	{attribute 'TcIecLibraryType'}
	{attribute 'external_name' := 'F_VN_SetAt_TcVnRectangle_DINT_GUID_35AC4059_132C_4AEE_E2AA_EA9A3D12C86B'}
	(* Sets the element at the specified index of the container. *)
	FUNCTION F_VN_SetAt_TcVnRectangle_DINT : HRESULT
	VAR_IN_OUT
		stElement	:	TcVnRectangle_DINT;	(* Element to set at the specified container position *)
	END_VAR
	VAR_INPUT
		ipContainer	:	ITcVnContainer;	(* Container with TcVnRectangle_DINT elements, in which the element at position nIndex is replaced by stElement *)
		nIndex	:	ULINT;	(* Index *)
		hrPrev	:	HRESULT;	(* HRESULT indicating the result of previous operations (If SUCCEEDED(hrPrev) equals false, no operation is executed.) *)
	END_VAR

END_FUNCTION

// Functions/Basic Container Operations/F_VN_SetAt/F_VN_SetAt_TcVnVector2_DINT

	{attribute 'TcIecLibraryType'}
	{attribute 'external_name' := 'F_VN_SetAt_TcVnVector2_DINT_GUID_5E02A515_5B29_40CA_DD70_70385858C65C'}
	(* Sets the element at the specified index of the container. *)
	FUNCTION F_VN_SetAt_TcVnVector2_DINT : HRESULT
	VAR_IN_OUT
		aElement	:	TcVnVector2_DINT;	(* Element to set at the specified container position *)
	END_VAR
	VAR_INPUT
		ipContainer	:	ITcVnContainer;	(* Container with TcVnVector2_DINT elements, in which the element at position nIndex is replaced by aElement *)
		nIndex	:	ULINT;	(* Index *)
		hrPrev	:	HRESULT;	(* HRESULT indicating the result of previous operations (If SUCCEEDED(hrPrev) equals false, no operation is executed.) *)
	END_VAR

END_FUNCTION

// Functions/Basic Container Operations/F_VN_SetAt/F_VN_SetAt_TcVnVector2_INT

	{attribute 'TcIecLibraryType'}
	{attribute 'external_name' := 'F_VN_SetAt_TcVnVector2_INT_GUID_9A54C8DF_EFEA_42F1_C006_DE70D5579EDC'}
	(* Sets the element at the specified index of the container. *)
	FUNCTION F_VN_SetAt_TcVnVector2_INT : HRESULT
	VAR_IN_OUT
		aElement	:	TcVnVector2_INT;	(* Element to set at the specified container position *)
	END_VAR
	VAR_INPUT
		ipContainer	:	ITcVnContainer;	(* Container with TcVnVector2_INT elements, in which the element at position nIndex is replaced by aElement *)
		nIndex	:	ULINT;	(* Index *)
		hrPrev	:	HRESULT;	(* HRESULT indicating the result of previous operations (If SUCCEEDED(hrPrev) equals false, no operation is executed.) *)
	END_VAR

END_FUNCTION

// Functions/Basic Container Operations/F_VN_SetAt/F_VN_SetAt_TcVnVector2_REAL

	{attribute 'TcIecLibraryType'}
	{attribute 'external_name' := 'F_VN_SetAt_TcVnVector2_REAL_GUID_8C701179_500E_467C_D95A_AFB507FC193B'}
	(* Sets the element at the specified index of the container. *)
	FUNCTION F_VN_SetAt_TcVnVector2_REAL : HRESULT
	VAR_IN_OUT
		aElement	:	TcVnVector2_REAL;	(* Element to set at the specified container position *)
	END_VAR
	VAR_INPUT
		ipContainer	:	ITcVnContainer;	(* Container with TcVnVector2_REAL elements, in which the element at position nIndex is replaced by aElement *)
		nIndex	:	ULINT;	(* Index *)
		hrPrev	:	HRESULT;	(* HRESULT indicating the result of previous operations (If SUCCEEDED(hrPrev) equals false, no operation is executed.) *)
	END_VAR

END_FUNCTION

// Functions/Basic Container Operations/F_VN_SetAt/F_VN_SetAt_TcVnVector2_SINT

	{attribute 'TcIecLibraryType'}
	{attribute 'external_name' := 'F_VN_SetAt_TcVnVector2_SINT_GUID_41E2A1B6_E23C_4E2B_F5BD_66BD8170D23F'}
	(* Sets the element at the specified index of the container. *)
	FUNCTION F_VN_SetAt_TcVnVector2_SINT : HRESULT
	VAR_IN_OUT
		aElement	:	TcVnVector2_SINT;	(* Element to set at the specified container position *)
	END_VAR
	VAR_INPUT
		ipContainer	:	ITcVnContainer;	(* Container with TcVnVector2_SINT elements, in which the element at position nIndex is replaced by aElement *)
		nIndex	:	ULINT;	(* Index *)
		hrPrev	:	HRESULT;	(* HRESULT indicating the result of previous operations (If SUCCEEDED(hrPrev) equals false, no operation is executed.) *)
	END_VAR

END_FUNCTION

// Functions/Basic Container Operations/F_VN_SetAt/F_VN_SetAt_TcVnVector2_UINT

	{attribute 'TcIecLibraryType'}
	{attribute 'external_name' := 'F_VN_SetAt_TcVnVector2_UINT_GUID_21FE93D3_4D33_43A5_D0AF_B50B4A89EE98'}
	(* Sets the element at the specified index of the container. *)
	FUNCTION F_VN_SetAt_TcVnVector2_UINT : HRESULT
	VAR_IN_OUT
		aElement	:	TcVnVector2_UINT;	(* Element to set at the specified container position *)
	END_VAR
	VAR_INPUT
		ipContainer	:	ITcVnContainer;	(* Container with TcVnVector2_UINT elements, in which the element at position nIndex is replaced by aElement *)
		nIndex	:	ULINT;	(* Index *)
		hrPrev	:	HRESULT;	(* HRESULT indicating the result of previous operations (If SUCCEEDED(hrPrev) equals false, no operation is executed.) *)
	END_VAR

END_FUNCTION

// Functions/Basic Container Operations/F_VN_SetAt/F_VN_SetAt_TcVnVector2_USINT

	{attribute 'TcIecLibraryType'}
	{attribute 'external_name' := 'F_VN_SetAt_TcVnVector2_USINT_GUID_71672D26_1D04_4018_CB62_849B8610E425'}
	(* Sets the element at the specified index of the container. *)
	FUNCTION F_VN_SetAt_TcVnVector2_USINT : HRESULT
	VAR_IN_OUT
		aElement	:	TcVnVector2_USINT;	(* Element to set at the specified container position *)
	END_VAR
	VAR_INPUT
		ipContainer	:	ITcVnContainer;	(* Container with TcVnVector2_USINT elements, in which the element at position nIndex is replaced by aElement *)
		nIndex	:	ULINT;	(* Index *)
		hrPrev	:	HRESULT;	(* HRESULT indicating the result of previous operations (If SUCCEEDED(hrPrev) equals false, no operation is executed.) *)
	END_VAR

END_FUNCTION

// Functions/Basic Container Operations/F_VN_SetAt/F_VN_SetAt_TcVnVector3_INT

	{attribute 'TcIecLibraryType'}
	{attribute 'external_name' := 'F_VN_SetAt_TcVnVector3_INT_GUID_B387FD7B_1A12_472C_FF84_9E1251FBA387'}
	(* Sets the element at the specified index of the container. *)
	FUNCTION F_VN_SetAt_TcVnVector3_INT : HRESULT
	VAR_IN_OUT
		aElement	:	TcVnVector3_INT;	(* Element to set at the specified container position *)
	END_VAR
	VAR_INPUT
		ipContainer	:	ITcVnContainer;	(* Container with TcVnVector3_INT elements, in which the element at position nIndex is replaced by aElement *)
		nIndex	:	ULINT;	(* Index *)
		hrPrev	:	HRESULT;	(* HRESULT indicating the result of previous operations (If SUCCEEDED(hrPrev) equals false, no operation is executed.) *)
	END_VAR

END_FUNCTION

// Functions/Basic Container Operations/F_VN_SetAt/F_VN_SetAt_TcVnVector3_REAL

	{attribute 'TcIecLibraryType'}
	{attribute 'external_name' := 'F_VN_SetAt_TcVnVector3_REAL_GUID_977FE56D_428C_427D_D95B_7AAACF1FD840'}
	(* Sets the element at the specified index of the container. *)
	FUNCTION F_VN_SetAt_TcVnVector3_REAL : HRESULT
	VAR_IN_OUT
		aElement	:	TcVnVector3_REAL;	(* Element to set at the specified container position *)
	END_VAR
	VAR_INPUT
		ipContainer	:	ITcVnContainer;	(* Container with TcVnVector3_REAL elements, in which the element at position nIndex is replaced by aElement *)
		nIndex	:	ULINT;	(* Index *)
		hrPrev	:	HRESULT;	(* HRESULT indicating the result of previous operations (If SUCCEEDED(hrPrev) equals false, no operation is executed.) *)
	END_VAR

END_FUNCTION

// Functions/Basic Container Operations/F_VN_SetAt/F_VN_SetAt_TcVnVector3_SINT

	{attribute 'TcIecLibraryType'}
	{attribute 'external_name' := 'F_VN_SetAt_TcVnVector3_SINT_GUID_82C45DC0_A60E_4C50_ED24_B824FCF78FFB'}
	(* Sets the element at the specified index of the container. *)
	FUNCTION F_VN_SetAt_TcVnVector3_SINT : HRESULT
	VAR_IN_OUT
		aElement	:	TcVnVector3_SINT;	(* Element to set at the specified container position *)
	END_VAR
	VAR_INPUT
		ipContainer	:	ITcVnContainer;	(* Container with TcVnVector3_SINT elements, in which the element at position nIndex is replaced by aElement *)
		nIndex	:	ULINT;	(* Index *)
		hrPrev	:	HRESULT;	(* HRESULT indicating the result of previous operations (If SUCCEEDED(hrPrev) equals false, no operation is executed.) *)
	END_VAR

END_FUNCTION

// Functions/Basic Container Operations/F_VN_SetAt/F_VN_SetAt_TcVnVector3_UINT

	{attribute 'TcIecLibraryType'}
	{attribute 'external_name' := 'F_VN_SetAt_TcVnVector3_UINT_GUID_B07401BC_3104_41A1_CD0F_B943A0C58B6B'}
	(* Sets the element at the specified index of the container. *)
	FUNCTION F_VN_SetAt_TcVnVector3_UINT : HRESULT
	VAR_IN_OUT
		aElement	:	TcVnVector3_UINT;	(* Element to set at the specified container position *)
	END_VAR
	VAR_INPUT
		ipContainer	:	ITcVnContainer;	(* Container with TcVnVector3_UINT elements, in which the element at position nIndex is replaced by aElement *)
		nIndex	:	ULINT;	(* Index *)
		hrPrev	:	HRESULT;	(* HRESULT indicating the result of previous operations (If SUCCEEDED(hrPrev) equals false, no operation is executed.) *)
	END_VAR

END_FUNCTION

// Functions/Basic Container Operations/F_VN_SetAt/F_VN_SetAt_TcVnVector3_USINT

	{attribute 'TcIecLibraryType'}
	{attribute 'external_name' := 'F_VN_SetAt_TcVnVector3_USINT_GUID_CA981836_58FF_4571_CBB8_6E1A27874793'}
	(* Sets the element at the specified index of the container. *)
	FUNCTION F_VN_SetAt_TcVnVector3_USINT : HRESULT
	VAR_IN_OUT
		aElement	:	TcVnVector3_USINT;	(* Element to set at the specified container position *)
	END_VAR
	VAR_INPUT
		ipContainer	:	ITcVnContainer;	(* Container with TcVnVector3_USINT elements, in which the element at position nIndex is replaced by aElement *)
		nIndex	:	ULINT;	(* Index *)
		hrPrev	:	HRESULT;	(* HRESULT indicating the result of previous operations (If SUCCEEDED(hrPrev) equals false, no operation is executed.) *)
	END_VAR

END_FUNCTION

// Functions/Basic Container Operations/F_VN_SetAt/F_VN_SetAt_TcVnVector4_DINT

	{attribute 'TcIecLibraryType'}
	{attribute 'external_name' := 'F_VN_SetAt_TcVnVector4_DINT_GUID_84075105_DF73_46B7_C61E_1F0647F1D871'}
	(* Sets the element at the specified index of the container. *)
	FUNCTION F_VN_SetAt_TcVnVector4_DINT : HRESULT
	VAR_IN_OUT
		aElement	:	TcVnVector4_DINT;	(* Element to set at the specified container position *)
	END_VAR
	VAR_INPUT
		ipContainer	:	ITcVnContainer;	(* Container with TcVnVector4_DINT elements, in which the element at position nIndex is replaced by aElement *)
		nIndex	:	ULINT;	(* Index *)
		hrPrev	:	HRESULT;	(* HRESULT indicating the result of previous operations (If SUCCEEDED(hrPrev) equals false, no operation is executed.) *)
	END_VAR

END_FUNCTION

// Functions/Basic Container Operations/F_VN_SetAt/F_VN_SetAt_TcVnVector4_INT

	{attribute 'TcIecLibraryType'}
	{attribute 'external_name' := 'F_VN_SetAt_TcVnVector4_INT_GUID_4C86CA39_B19A_4E94_C5DE_D1DC020F94C8'}
	(* Sets the element at the specified index of the container. *)
	FUNCTION F_VN_SetAt_TcVnVector4_INT : HRESULT
	VAR_IN_OUT
		aElement	:	TcVnVector4_INT;	(* Element to set at the specified container position *)
	END_VAR
	VAR_INPUT
		ipContainer	:	ITcVnContainer;	(* Container with TcVnVector4_INT elements, in which the element at position nIndex is replaced by aElement *)
		nIndex	:	ULINT;	(* Index *)
		hrPrev	:	HRESULT;	(* HRESULT indicating the result of previous operations (If SUCCEEDED(hrPrev) equals false, no operation is executed.) *)
	END_VAR

END_FUNCTION

// Functions/Basic Container Operations/F_VN_SetAt/F_VN_SetAt_TcVnVector4_LREAL

	{attribute 'TcIecLibraryType'}
	{attribute 'external_name' := 'F_VN_SetAt_TcVnVector4_LREAL_GUID_B3814A00_38B2_4F72_CE05_8FB87EDAF63D'}
	(* Sets the element at the specified index of the container. *)
	FUNCTION F_VN_SetAt_TcVnVector4_LREAL : HRESULT
	VAR_IN_OUT
		aElement	:	TcVnVector4_LREAL;	(* Element to set at the specified container position *)
	END_VAR
	VAR_INPUT
		ipContainer	:	ITcVnContainer;	(* Container with TcVnVector4_LREAL elements, in which the element at position nIndex is replaced by aElement *)
		nIndex	:	ULINT;	(* Index *)
		hrPrev	:	HRESULT;	(* HRESULT indicating the result of previous operations (If SUCCEEDED(hrPrev) equals false, no operation is executed.) *)
	END_VAR

END_FUNCTION

// Functions/Basic Container Operations/F_VN_SetAt/F_VN_SetAt_TcVnVector4_REAL

	{attribute 'TcIecLibraryType'}
	{attribute 'external_name' := 'F_VN_SetAt_TcVnVector4_REAL_GUID_64AEDC0F_5778_44DB_ECE6_E811B6DE732F'}
	(* Sets the element at the specified index of the container. *)
	FUNCTION F_VN_SetAt_TcVnVector4_REAL : HRESULT
	VAR_IN_OUT
		aElement	:	TcVnVector4_REAL;	(* Element to set at the specified container position *)
	END_VAR
	VAR_INPUT
		ipContainer	:	ITcVnContainer;	(* Container with TcVnVector4_REAL elements, in which the element at position nIndex is replaced by aElement *)
		nIndex	:	ULINT;	(* Index *)
		hrPrev	:	HRESULT;	(* HRESULT indicating the result of previous operations (If SUCCEEDED(hrPrev) equals false, no operation is executed.) *)
	END_VAR

END_FUNCTION

// Functions/Basic Container Operations/F_VN_SetAt/F_VN_SetAt_TcVnVector4_SINT

	{attribute 'TcIecLibraryType'}
	{attribute 'external_name' := 'F_VN_SetAt_TcVnVector4_SINT_GUID_9A249CC5_D1EE_48B3_F4D3_D6345D13532B'}
	(* Sets the element at the specified index of the container. *)
	FUNCTION F_VN_SetAt_TcVnVector4_SINT : HRESULT
	VAR_IN_OUT
		aElement	:	TcVnVector4_SINT;	(* Element to set at the specified container position *)
	END_VAR
	VAR_INPUT
		ipContainer	:	ITcVnContainer;	(* Container with TcVnVector4_SINT elements, in which the element at position nIndex is replaced by aElement *)
		nIndex	:	ULINT;	(* Index *)
		hrPrev	:	HRESULT;	(* HRESULT indicating the result of previous operations (If SUCCEEDED(hrPrev) equals false, no operation is executed.) *)
	END_VAR

END_FUNCTION

// Functions/Basic Container Operations/F_VN_SetAt/F_VN_SetAt_TcVnVector4_UINT

	{attribute 'TcIecLibraryType'}
	{attribute 'external_name' := 'F_VN_SetAt_TcVnVector4_UINT_GUID_9C7C3011_85A8_431A_EEDE_04346BDEC621'}
	(* Sets the element at the specified index of the container. *)
	FUNCTION F_VN_SetAt_TcVnVector4_UINT : HRESULT
	VAR_IN_OUT
		aElement	:	TcVnVector4_UINT;	(* Element to set at the specified container position *)
	END_VAR
	VAR_INPUT
		ipContainer	:	ITcVnContainer;	(* Container with TcVnVector4_UINT elements, in which the element at position nIndex is replaced by aElement *)
		nIndex	:	ULINT;	(* Index *)
		hrPrev	:	HRESULT;	(* HRESULT indicating the result of previous operations (If SUCCEEDED(hrPrev) equals false, no operation is executed.) *)
	END_VAR

END_FUNCTION

// Functions/Basic Container Operations/F_VN_SetAt/F_VN_SetAt_TcVnVector4_USINT

	{attribute 'TcIecLibraryType'}
	{attribute 'external_name' := 'F_VN_SetAt_TcVnVector4_USINT_GUID_8CCBCF1A_6BF1_414F_D7CE_FA6418BF3A5A'}
	(* Sets the element at the specified index of the container. *)
	FUNCTION F_VN_SetAt_TcVnVector4_USINT : HRESULT
	VAR_IN_OUT
		aElement	:	TcVnVector4_USINT;	(* Element to set at the specified container position *)
	END_VAR
	VAR_INPUT
		ipContainer	:	ITcVnContainer;	(* Container with TcVnVector4_USINT elements, in which the element at position nIndex is replaced by aElement *)
		nIndex	:	ULINT;	(* Index *)
		hrPrev	:	HRESULT;	(* HRESULT indicating the result of previous operations (If SUCCEEDED(hrPrev) equals false, no operation is executed.) *)
	END_VAR

END_FUNCTION

// Functions/Basic Container Operations/F_VN_SetAt/F_VN_SetAt_UDINT

	{attribute 'TcIecLibraryType'}
	{attribute 'external_name' := 'F_VN_SetAt_UDINT_GUID_C39B4E59_D3B2_44DA_C04B_593E8FE83763'}
	(* Sets the element at the specified index of the container. *)
	FUNCTION F_VN_SetAt_UDINT : HRESULT
	VAR_INPUT
		nElement	:	UDINT;	(* Element to set at the specified container position *)
		ipContainer	:	ITcVnContainer;	(* Container with UDINT elements, in which the element at position nIndex is replaced by nElement *)
		nIndex	:	ULINT;	(* Index *)
		hrPrev	:	HRESULT;	(* HRESULT indicating the result of previous operations (If SUCCEEDED(hrPrev) equals false, no operation is executed.) *)
	END_VAR

END_FUNCTION

// Functions/Basic Container Operations/F_VN_SetAt/F_VN_SetAt_UINT

	{attribute 'TcIecLibraryType'}
	{attribute 'external_name' := 'F_VN_SetAt_UINT_GUID_973D05B9_94F7_4B2D_E393_23B939525C18'}
	(* Sets the element at the specified index of the container. *)
	FUNCTION F_VN_SetAt_UINT : HRESULT
	VAR_INPUT
		nElement	:	UINT;	(* Element to set at the specified container position *)
		ipContainer	:	ITcVnContainer;	(* Container with UINT elements, in which the element at position nIndex is replaced by nElement *)
		nIndex	:	ULINT;	(* Index *)
		hrPrev	:	HRESULT;	(* HRESULT indicating the result of previous operations (If SUCCEEDED(hrPrev) equals false, no operation is executed.) *)
	END_VAR

END_FUNCTION

// Functions/Basic Container Operations/F_VN_SetAt/F_VN_SetAt_ULINT

	{attribute 'TcIecLibraryType'}
	{attribute 'external_name' := 'F_VN_SetAt_ULINT_GUID_FC881A2A_C368_47AC_FDE8_4603A11A5BED'}
	(* Sets the element at the specified index of the container. *)
	FUNCTION F_VN_SetAt_ULINT : HRESULT
	VAR_INPUT
		nElement	:	ULINT;	(* Element to set at the specified container position *)
		ipContainer	:	ITcVnContainer;	(* Container with ULINT elements, in which the element at position nIndex is replaced by nElement *)
		nIndex	:	ULINT;	(* Index *)
		hrPrev	:	HRESULT;	(* HRESULT indicating the result of previous operations (If SUCCEEDED(hrPrev) equals false, no operation is executed.) *)
	END_VAR

END_FUNCTION

// Functions/Basic Container Operations/F_VN_SetAt/F_VN_SetAt_USINT

	{attribute 'TcIecLibraryType'}
	{attribute 'external_name' := 'F_VN_SetAt_USINT_GUID_71675C04_000B_40FA_E123_CBE4050ACA90'}
	(* Sets the element at the specified index of the container. *)
	FUNCTION F_VN_SetAt_USINT : HRESULT
	VAR_INPUT
		nElement	:	USINT;	(* Element to set at the specified container position *)
		ipContainer	:	ITcVnContainer;	(* Container with USINT elements, in which the element at position nIndex is replaced by nElement *)
		nIndex	:	ULINT;	(* Index *)
		hrPrev	:	HRESULT;	(* HRESULT indicating the result of previous operations (If SUCCEEDED(hrPrev) equals false, no operation is executed.) *)
	END_VAR

END_FUNCTION

// Functions/Geometric and Coordinate Transformations/Calibration/F_VN_CalibrateCamera

	{attribute 'TcIecLibraryType'}
	{attribute 'external_name' := 'F_VN_CalibrateCamera_GUID_EBB15309_7B02_4BBD_EDF8_3E60282ECCFA'}
	(* Compute the camera parameters (intrinsic + extrinsic) by evaluating an image containing a calibration pattern (circles). *)
	FUNCTION F_VN_CalibrateCamera : HRESULT
	VAR_INPUT
		ipSrcImage	:	ITcVnImage;	(* Source image containing a calibration pattern (1 channel, USINT elements) *)
		ipReferencePoints	:	ITcVnContainer;	(* Reference calibration pattern point positions (ContainerType_Vector_TcVnPoint3_REAL) *)
	END_VAR
	VAR_IN_OUT
		aCameraMatrix	:	TcVnMatrix3x3_LREAL;	(* Returns the camera matrix *)
		aDistortionCoefficients	:	TcVnArray8_LREAL;	(* Returns the lens distortion coefficients [k1, k2, p1, p2, k3, k4, k5, k6] *)
		aRotationMatrix	:	TcVnMatrix3x3_LREAL;	(* Returns the rotation matrix *)
		aTranslationVector	:	TcVnVector3_LREAL;	(* Returns the translation vector *)
		fReprojError	:	LREAL;	(* Returns the reprojection error *)
		stBlobDetectionParams	:	TcVnParamsBlobDetection;	(* Parameters for the internally used F_VN_DetectBlobs function *)
		stCalibrationOptions	:	TcVnCameraCalibrationOptions;	(* Calibration options *)
	END_VAR
	VAR_INPUT
		hrPrev	:	HRESULT;	(* HRESULT indicating the result of previous operations (If SUCCEEDED(hrPrev) equals false, no operation is executed.) *)
	END_VAR

END_FUNCTION

// Functions/Geometric and Coordinate Transformations/Calibration/F_VN_CalibrateCameraExp

	{attribute 'TcIecLibraryType'}
	{attribute 'external_name' := 'F_VN_CalibrateCameraExp_GUID_1D6493E0_8C99_44E7_F620_1AFFF7BB97DC'}
	(* Compute the camera parameters (intrinsic + extrinsic) by evaluating images containing a calibration pattern (circles). The extrinsic parameters are computed for the first image in the array. (expert function) *)
	FUNCTION F_VN_CalibrateCameraExp : HRESULT
	VAR_INPUT
		pSrcImages	:	PVOID;	(* Pointer to an array of source images, each containing the same calibration pattern (1 channel, USINT elements) *)
		nSrcArraySize	:	UINT;	(* pSrcImages array size *)
		ipReferencePoints	:	ITcVnContainer;	(* Reference calibration pattern point positions (ContainerType_Vector_TcVnPoint3_REAL) *)
	END_VAR
	VAR_IN_OUT
		aCameraMatrix	:	TcVnMatrix3x3_LREAL;	(* Returns the camera matrix *)
		aDistortionCoefficients	:	TcVnArray8_LREAL;	(* Returns the lens distortion coefficients [k1, k2, p1, p2, k3, k4, k5, k6] *)
		aRotationMatrix	:	TcVnMatrix3x3_LREAL;	(* Returns the rotation matrix *)
		aTranslationVector	:	TcVnVector3_LREAL;	(* Returns the translation vector *)
		fReprojError	:	LREAL;	(* Returns the reprojection error *)
		stBlobDetectionParams	:	TcVnParamsBlobDetection;	(* Parameters for the internally used F_VN_DetectBlobs function *)
		stCalibrationOptions	:	TcVnCameraCalibrationOptions;	(* Calibration options *)
	END_VAR
	VAR_INPUT
		hrPrev	:	HRESULT;	(* HRESULT indicating the result of previous operations (If SUCCEEDED(hrPrev) equals false, no operation is executed.) *)
	END_VAR

END_FUNCTION

// Functions/Geometric and Coordinate Transformations/Calibration/F_VN_CalibrateCameraExp2

	{attribute 'TcIecLibraryType'}
	{attribute 'external_name' := 'F_VN_CalibrateCameraExp2_GUID_8981380C_F1D9_4601_D366_FF624EB09033'}
	(* Compute the camera parameters (intrinsic + extrinsic) by evaluating images containing a calibration pattern (circles). The extrinsic parameters are computed for the first image in the array. (expert function) *)
	FUNCTION F_VN_CalibrateCameraExp2 : HRESULT
	VAR_INPUT
		pSrcImages	:	PVOID;	(* Pointer to an array of source images, each containing the same calibration pattern (1 channel, USINT elements) *)
		nSrcArraySize	:	UINT;	(* pSrcImages array size *)
		ipReferencePoints	:	ITcVnContainer;	(* Reference calibration pattern point positions (ContainerType_Vector_TcVnPoint3_REAL) *)
	END_VAR
	VAR_IN_OUT
		aCameraMatrix	:	TcVnMatrix3x3_LREAL;	(* Returns the camera matrix *)
		aDistortionCoefficients	:	TcVnArray8_LREAL;	(* Returns the lens distortion coefficients [k1, k2, p1, p2, k3, k4, k5, k6] *)
		aRotationMatrix	:	TcVnMatrix3x3_LREAL;	(* Returns the rotation matrix *)
		aTranslationVector	:	TcVnVector3_LREAL;	(* Returns the translation vector *)
		fReprojError	:	LREAL;	(* Returns the reprojection error *)
		stBlobDetectionParams	:	TcVnParamsBlobDetection;	(* Parameters for the internally used F_VN_DetectBlobs function *)
		stCalibrationOptions	:	TcVnCameraCalibrationOptions;	(* Calibration options *)
	END_VAR
	VAR_INPUT
		bSubpixelAccuracy	:	BOOL;	(* If true, the pattern points are detected with subpixel accuracy *)
		eEdgeDirection	:	ETcVnEdgeDirection;	(* Specification of the edge direction to search for (from center to outside ellipse) *)
		fMinStrength	:	REAL;	(* Specification of the minimum strength (intensity difference) of the edge to search for *)
		nMaxThickness	:	UDINT;	(* Specification of the maximum thickness of the edge to search for, which means fMinStrength must be reached within nMaxThickness pixels *)
		nSubpixelsIterations	:	UDINT;	(* Specifies the number of subpixels (for INTERPOLATION, 10 - 20 usually is sufficient) or maximum number of iterations for optimizing the parameters (for APPROX_ERF and APPROX_GAUSSIAN, 50 - 100 usually is sufficient) *)
		nSearchLines	:	UDINT;	(* Specifies the amount of search lines, which are equally distributed in all directions (must be >= 8 and a multiple of 4) *)
		fApproxPrecision	:	REAL;	(* Specifies the approximation precision for APPROX_ERF and APPROX_GAUSSIAN (0.001 usually is sufficient, unused for INTERPOLATION) *)
		eAlgorithm	:	ETcVnEdgeDetectionAlgorithm;	(* Selection of the edge detection algorithm *)
		hrPrev	:	HRESULT;	(* HRESULT indicating the result of previous operations (If SUCCEEDED(hrPrev) equals false, no operation is executed.) *)
	END_VAR

END_FUNCTION

// Functions/Geometric and Coordinate Transformations/Calibration/F_VN_CalibrateCameraExp3

	{attribute 'TcIecLibraryType'}
	{attribute 'external_name' := 'F_VN_CalibrateCameraExp3_GUID_D9F3CD5D_1398_4870_FF18_533CD0366399'}
	(* Compute the camera parameters (intrinsic + extrinsic) by evaluating images containing a calibration pattern (circles). The extrinsic parameters are computed for the first image in the array. (expert function) *)
	FUNCTION F_VN_CalibrateCameraExp3 : HRESULT
	VAR_INPUT
		pSrcImages	:	PVOID;	(* Pointer to an array of source images, each containing the same calibration pattern (1 channel, USINT elements) *)
		nSrcArraySize	:	UINT;	(* pSrcImages array size *)
		ipReferencePoints	:	ITcVnContainer;	(* Reference calibration pattern point positions (ContainerType_Vector_TcVnPoint3_REAL) *)
	END_VAR
	VAR_IN_OUT
		aCameraMatrix	:	TcVnMatrix3x3_LREAL;	(* Returns the camera matrix *)
		aDistortionCoefficients	:	TcVnArray8_LREAL;	(* Returns the lens distortion coefficients [k1, k2, p1, p2, k3, k4, k5, k6] *)
		aRotationMatrix	:	TcVnMatrix3x3_LREAL;	(* Returns the rotation matrix *)
		aTranslationVector	:	TcVnVector3_LREAL;	(* Returns the translation vector *)
		fReprojError	:	LREAL;	(* Returns the reprojection error *)
		stBlobDetectionParams	:	TcVnParamsBlobDetection;	(* Parameters for the internally used F_VN_DetectBlobs function *)
		stCalibrationOptions	:	TcVnCameraCalibrationOptions;	(* Calibration options *)
	END_VAR
	VAR_INPUT
		bSubpixelAccuracy	:	BOOL;	(* If true, the pattern points are detected with subpixel accuracy *)
		eEdgeDirection	:	ETcVnEdgeDirection;	(* Specification of the edge direction to search for (from center to outside ellipse) *)
		fMinStrength	:	REAL;	(* Specification of the minimum strength (intensity difference) of the edge to search for *)
		nMaxThickness	:	UDINT;	(* Specification of the maximum thickness of the edge to search for, which means fMinStrength must be reached within nMaxThickness pixels *)
		nSubpixelsIterations	:	UDINT;	(* Specifies the number of subpixels (for INTERPOLATION, 10 - 20 usually is sufficient) or maximum number of iterations for optimizing the parameters (for APPROX_ERF and APPROX_GAUSSIAN, 50 - 100 usually is sufficient) *)
		nSearchLines	:	UDINT;	(* Specifies the amount of search lines, which are equally distributed in all directions (must be >= 8 and a multiple of 4) *)
		fApproxPrecision	:	REAL;	(* Specifies the approximation precision for APPROX_ERF and APPROX_GAUSSIAN (0.001 usually is sufficient, unused for INTERPOLATION) *)
		eAlgorithm	:	ETcVnEdgeDetectionAlgorithm;	(* Selection of the edge detection algorithm *)
		eWorldSystem	:	ETcVnWorldCoordinateSystem;	(* World coordinate system orientation *)
		hrPrev	:	HRESULT;	(* HRESULT indicating the result of previous operations (If SUCCEEDED(hrPrev) equals false, no operation is executed.) *)
	END_VAR

END_FUNCTION

// Functions/Geometric and Coordinate Transformations/Calibration/F_VN_CalibrateCameraManually

	{attribute 'TcIecLibraryType'}
	{attribute 'external_name' := 'F_VN_CalibrateCameraManually_GUID_5DA30166_3B16_4F1A_EA40_4DD63022F860'}
	(* Compute the camera parameters (intrinsic + extrinsic). The extrinsic parameters are computed for the first inner container. *)
	FUNCTION F_VN_CalibrateCameraManually : HRESULT
	VAR_INPUT
		ipImagePoints	:	ITcVnContainer;	(* Provided image points of multiple images (ContainerType_Vector_Vector_TcVnPoint2_REAL, each inner container with at least 6 points). The container and point order must match ipReferencePoints. *)
		nImageWidth	:	UDINT;	(* Image width *)
		nImageHeight	:	UDINT;	(* Image height *)
		ipReferencePoints	:	ITcVnContainer;	(* Reference world points (ContainerType_Vector_Vector_TcVnPoint3_REAL). The number of inner containers and their amount of points must match ipImagePoints. *)
	END_VAR
	VAR_IN_OUT
		aCameraMatrix	:	TcVnMatrix3x3_LREAL;	(* Returns the camera matrix *)
		aDistortionCoefficients	:	TcVnArray8_LREAL;	(* Returns the lens distortion coefficients [k1, k2, p1, p2, k3, k4, k5, k6] *)
		aRotationMatrix	:	TcVnMatrix3x3_LREAL;	(* Returns the rotation matrix (for the first inner container) *)
		aTranslationVector	:	TcVnVector3_LREAL;	(* Returns the translation vector (for the first inner container) *)
		fReprojError	:	LREAL;	(* Returns the reprojection error *)
		stCalibrationOptions	:	TcVnCameraCalibrationOptions;	(* Calibration options *)
	END_VAR
	VAR_INPUT
		hrPrev	:	HRESULT;	(* HRESULT indicating the result of previous operations (If SUCCEEDED(hrPrev) equals false, no operation is executed.) *)
	END_VAR

END_FUNCTION

// Functions/Geometric and Coordinate Transformations/Calibration/F_VN_CalibrateCameraManuallyExp

	{attribute 'TcIecLibraryType'}
	{attribute 'external_name' := 'F_VN_CalibrateCameraManuallyExp_GUID_DECD6B85_89B7_4630_E66B_3B96B0529CB2'}
	(* Compute the camera parameters (intrinsic + extrinsic). The extrinsic parameters are computed for the first inner container. (expert function) *)
	FUNCTION F_VN_CalibrateCameraManuallyExp : HRESULT
	VAR_INPUT
		ipImagePoints	:	ITcVnContainer;	(* Provided image points of multiple images (ContainerType_Vector_Vector_TcVnPoint2_REAL, each inner container with at least 6 points). The container and point order must match ipReferencePoints. *)
		nImageWidth	:	UDINT;	(* Image width *)
		nImageHeight	:	UDINT;	(* Image height *)
		ipReferencePoints	:	ITcVnContainer;	(* Reference world points (ContainerType_Vector_Vector_TcVnPoint3_REAL). The number of inner containers and their amount of points must match ipImagePoints. *)
	END_VAR
	VAR_IN_OUT
		aCameraMatrix	:	TcVnMatrix3x3_LREAL;	(* Returns the camera matrix *)
		aDistortionCoefficients	:	TcVnArray8_LREAL;	(* Returns the lens distortion coefficients [k1, k2, p1, p2, k3, k4, k5, k6] *)
		aRotationMatrix	:	TcVnMatrix3x3_LREAL;	(* Returns the rotation matrix (for the first inner container) *)
		aTranslationVector	:	TcVnVector3_LREAL;	(* Returns the translation vector (for the first inner container) *)
		fReprojError	:	LREAL;	(* Returns the reprojection error *)
		stCalibrationOptions	:	TcVnCameraCalibrationOptions;	(* Calibration options *)
	END_VAR
	VAR_INPUT
		eWorldSystem	:	ETcVnWorldCoordinateSystem;	(* World coordinate system orientation *)
		hrPrev	:	HRESULT;	(* HRESULT indicating the result of previous operations (If SUCCEEDED(hrPrev) equals false, no operation is executed.) *)
	END_VAR

END_FUNCTION

// Functions/Geometric and Coordinate Transformations/Calibration/F_VN_CalibrateCameraPlanar

	{attribute 'TcIecLibraryType'}
	{attribute 'external_name' := 'F_VN_CalibrateCameraPlanar_GUID_DD8D0D8C_ACE8_4133_C290_06DF72655118'}
	(* Calibrate camera using a planar calibration pattern comprised of four circles marking the corners of a rectangle. *)
	FUNCTION F_VN_CalibrateCameraPlanar : HRESULT
	VAR_INPUT
		ipSrcImage	:	ITcVnImage;	(* Binary source image (background zero, markers non-zero) *)
	END_VAR
	VAR_IN_OUT
		aMarkerPositions	:	TcVnArray4_Point2_REAL;	(* Marker positions within their plane using world units (right-handed coordinate system) *)
		aTransformationMatrix	:	TcVnMatrix3x3_LREAL;	(* Returns a 3-by-3 matrix for the transformation from image coordinates into the reference coordinate system *)
	END_VAR
	VAR_INPUT
		hrPrev	:	HRESULT;	(* HRESULT indicating the result of previous operations (If SUCCEEDED(hrPrev) equals false, no operation is executed.) *)
	END_VAR

END_FUNCTION

// Functions/Geometric and Coordinate Transformations/Calibration/F_VN_CalibrateCameraPlanarExp

	{attribute 'TcIecLibraryType'}
	{attribute 'external_name' := 'F_VN_CalibrateCameraPlanarExp_GUID_7DEAD94E_63B2_4C34_D746_EB385A5F99A0'}
	(* Calibrate camera using a planar calibration pattern comprised of four circles marking the corners of a rectangle. (expert function) *)
	FUNCTION F_VN_CalibrateCameraPlanarExp : HRESULT
	VAR_INPUT
		ipSrcImage	:	ITcVnImage;	(* Binary source image (background zero, markers non-zero) *)
	END_VAR
	VAR_IN_OUT
		aMarkerPositions	:	TcVnArray4_Point2_REAL;	(* Marker positions within their plane using world units (right-handed coordinate system) *)
		aTransformationMatrix	:	TcVnMatrix3x3_LREAL;	(* Returns a 3-by-3 matrix for the transformation from image coordinates into the reference coordinate system *)
		aMarkerImagePositions	:	TcVnArray4_Point2_REAL;	(* Returns the marker positions in image coordinates (left-handed coordinate system) *)
	END_VAR
	VAR_INPUT
		nMinMarkerArea	:	UDINT;	(* Minimum area for the detection of markers (Smaller markers are ignored.) *)
		nMaxMarkerArea	:	UDINT;	(* Maximum area for the detection of markers (Larger markers are ignored.) *)
		fMaxMarkerEccentricity	:	LREAL;	(* Maximum eccenticity for the detection of markers (The eccentricity measures deviations from a round shape (eccentricity = 0: round object; eccentricity = 1.0:  linear object).) *)
		hrPrev	:	HRESULT;	(* HRESULT indicating the result of previous operations (If SUCCEEDED(hrPrev) equals false, no operation is executed.) *)
	END_VAR

END_FUNCTION

// Functions/Geometric and Coordinate Transformations/Calibration/F_VN_CalibrateLinescanCamera

	{attribute 'TcIecLibraryType'}
	{attribute 'external_name' := 'F_VN_CalibrateLinescanCamera_GUID_800BBE18_64E6_4C93_C932_85B991825405'}
	(* Compute the camera parameters (intrinsic + extrinsic) by evaluating images containing a line calibration pattern. The pattern must consist of alternating vertical and diagonal lines, with each diagonal having the same constant slope: |\|\|...\|. The results are only valid for the x-direction of a line scan image. To get accurate x-values for a transformation into world coordinates, the y-coordinate must be set to half the sensor width and so equal to the cy-value of the camera matrix. For other y-values, the results are approximated and can be inaccurate. The extrinsic parameters are computed for the first image in the array. *)
	FUNCTION F_VN_CalibrateLinescanCamera : HRESULT
	VAR_INPUT
		pSrcImages	:	PVOID;	(* Pointer to an array of 1 or more source images (1 channel). If the images have more than 1 row, each row must contain an image of the same pattern position. *)
		nSrcArraySize	:	UINT;	(* pSrcImages array size *)
		ipPatternLineOrigins	:	ITcVnContainer;	(* X position of the pattern line origins (ContainerType_Vector_REAL, usually same origin for vertical and following diagonal line) *)
		fSlopeRad	:	LREAL;	(* Slope of the diagonal line in rad (> 0, < PI/2), relative to the vertical line (i.e., 0 would be a vertical line, PI/2 a horizontal line) *)
	END_VAR
	VAR_IN_OUT
		aCameraMatrix	:	TcVnMatrix3x3_LREAL;	(* Returns the camera matrix *)
		aDistortionCoefficients	:	TcVnArray8_LREAL;	(* Returns the lens distortion coefficients [k1, k2, p1, p2, k3, k4, k5, k6] *)
		aRotationMatrix	:	TcVnMatrix3x3_LREAL;	(* Returns the rotation matrix *)
		aTranslationVector	:	TcVnVector3_LREAL;	(* Returns the translation vector *)
		fReprojError	:	LREAL;	(* Returns the reprojection error *)
		stCalibrationOptions	:	TcVnCameraCalibrationOptions;	(* Calibration options (recommended to set bFixAspectRatio, bFixPrincipalPoint, bZeroTangentDist) *)
	END_VAR
	VAR_INPUT
		eEdgeDirection	:	ETcVnEdgeDirection;	(* Specification of the edge direction to search for *)
		hrPrev	:	HRESULT;	(* HRESULT indicating the result of previous operations (If SUCCEEDED(hrPrev) equals false, no operation is executed.) *)
	END_VAR

END_FUNCTION

// Functions/Geometric and Coordinate Transformations/Calibration/F_VN_CalibrateLinescanCameraExp

	{attribute 'TcIecLibraryType'}
	{attribute 'external_name' := 'F_VN_CalibrateLinescanCameraExp_GUID_AD67159F_52AC_4940_E181_6CB9805B9B64'}
	(* Compute the camera parameters (intrinsic + extrinsic) by evaluating images containing a line calibration pattern. The pattern must consist of alternating vertical and diagonal lines, with each diagonal having the same constant slope: |\|\|...\|. The results are only valid for the x-direction of a line scan image. To get accurate x-values for a transformation into world coordinates, the y-coordinate must be set to half the sensor width and so equal to the cy-value of the camera matrix. For other y-values, the results are approximated and can be inaccurate. The extrinsic parameters are computed for the first image in the array. (expert function) *)
	FUNCTION F_VN_CalibrateLinescanCameraExp : HRESULT
	VAR_INPUT
		pSrcImages	:	PVOID;	(* Pointer to an array of 1 or more source images (1 channel). If the images have more than 1 row, each row must contain an image of the same pattern position. *)
		nSrcArraySize	:	UINT;	(* pSrcImages array size *)
		ipPatternLineOrigins	:	ITcVnContainer;	(* X position of the pattern line origins (ContainerType_Vector_REAL, usually same origin for vertical and following diagonal line) *)
		fSlopeRad	:	LREAL;	(* Slope of the diagonal line in rad (> 0, < PI/2), relative to the vertical line (i.e., 0 would be a vertical line, PI/2 a horizontal line) *)
	END_VAR
	VAR_IN_OUT
		aCameraMatrix	:	TcVnMatrix3x3_LREAL;	(* Returns the camera matrix *)
		aDistortionCoefficients	:	TcVnArray8_LREAL;	(* Returns the lens distortion coefficients [k1, k2, p1, p2, k3, k4, k5, k6] *)
		aRotationMatrix	:	TcVnMatrix3x3_LREAL;	(* Returns the rotation matrix *)
		aTranslationVector	:	TcVnVector3_LREAL;	(* Returns the translation vector *)
		fReprojError	:	LREAL;	(* Returns the reprojection error *)
		stCalibrationOptions	:	TcVnCameraCalibrationOptions;	(* Calibration options (recommended to set bFixAspectRatio, bFixPrincipalPoint, bZeroTangentDist) *)
	END_VAR
	VAR_INPUT
		eEdgeDirection	:	ETcVnEdgeDirection;	(* Specification of the edge direction to search for *)
		fMinStrength	:	REAL;	(* Specification of the minimum strength (intensity difference) of the edge to search for *)
		nMaxSearchLines	:	UDINT;	(* Maximum number of search lines (equally distributed over the image height, at most 1 searchline per image row) *)
		nMaxThickness	:	UDINT;	(* Specification of the maximum thickness of the edge to search for, which means fMinStrength must be reached within nMaxThickness pixels *)
		nSubpixelsIterations	:	UDINT;	(* Specifies the number of subpixels (for INTERPOLATION, 10 - 20 usually is sufficient) or maximum number of iterations for optimizing the parameters (for APPROX_ERF and APPROX_GAUSSIAN, 50 - 100 usually is sufficient) *)
		fApproxPrecision	:	REAL;	(* Specifies the approximation precision for APPROX_ERF and APPROX_GAUSSIAN (0.001 usually is sufficient, unused for INTERPOLATION) *)
		eAlgorithm	:	ETcVnEdgeDetectionAlgorithm;	(* Selection of the edge detection algorithm *)
		hrPrev	:	HRESULT;	(* HRESULT indicating the result of previous operations (If SUCCEEDED(hrPrev) equals false, no operation is executed.) *)
	END_VAR

END_FUNCTION

// Functions/Geometric and Coordinate Transformations/Calibration/F_VN_CompensateLensDistortion

	{attribute 'TcIecLibraryType'}
	{attribute 'external_name' := 'F_VN_CompensateLensDistortion_GUID_489AFC10_366F_422A_FEA8_C663F90A1CC1'}
	(* Transforms an image to compensate the lens distortion. *)
	FUNCTION F_VN_CompensateLensDistortion : HRESULT
	VAR_INPUT
		ipSrcImage	:	ITcVnImage;	(* Source image *)
		ipDestImage	:	REFERENCE TO ITcVnImage;	(* Destination image (An appropriate destination image will be created if required.) *)
	END_VAR
	VAR_IN_OUT
		aCameraMatrix	:	TcVnMatrix3x3_LREAL;	(* Camera matrix containing the intrinsic parameters *)
		aDistortionCoefficients	:	TcVnArray4_LREAL;	(* Lens distortion coefficients [k1, k2, p1, p2] *)
	END_VAR
	VAR_INPUT
		hrPrev	:	HRESULT;	(* HRESULT indicating the result of previous operations (If SUCCEEDED(hrPrev) equals false, no operation is executed.) *)
	END_VAR

END_FUNCTION

// Functions/Geometric and Coordinate Transformations/Calibration/F_VN_CompensateLensDistortionExp1

	{attribute 'TcIecLibraryType'}
	{attribute 'external_name' := 'F_VN_CompensateLensDistortionExp1_GUID_D2E79A17_6A4C_4E31_F93C_D1A6B8522041'}
	(* Transforms an image to compensate the lens distortion. (expert function) *)
	FUNCTION F_VN_CompensateLensDistortionExp1 : HRESULT
	VAR_INPUT
		ipSrcImage	:	ITcVnImage;	(* Source image *)
		ipDestImage	:	REFERENCE TO ITcVnImage;	(* Destination image (An appropriate destination image will be created if required.) *)
	END_VAR
	VAR_IN_OUT
		aCameraMatrix	:	TcVnMatrix3x3_LREAL;	(* Camera matrix containing the intrinsic parameters *)
		aDistortionCoefficients	:	TcVnArray8_LREAL;	(* Lens distortion coefficients [k1, k2, p1, p2, k3, k4, k5, k6] *)
	END_VAR
	VAR_INPUT
		hrPrev	:	HRESULT;	(* HRESULT indicating the result of previous operations (If SUCCEEDED(hrPrev) equals false, no operation is executed.) *)
	END_VAR

END_FUNCTION

// Functions/Geometric and Coordinate Transformations/Calibration/F_VN_CompensateLensDistortionExp2

	{attribute 'TcIecLibraryType'}
	{attribute 'external_name' := 'F_VN_CompensateLensDistortionExp2_GUID_2D7CC59B_2F49_4E33_DD38_7EA1C5FBDC31'}
	(* Transforms an image to compensate the lens distortion. (expert function) *)
	FUNCTION F_VN_CompensateLensDistortionExp2 : HRESULT
	VAR_INPUT
		ipSrcImage	:	ITcVnImage;	(* Source image *)
		ipDestImage	:	REFERENCE TO ITcVnImage;	(* Destination image (An appropriate destination image will be created if required.) *)
	END_VAR
	VAR_IN_OUT
		aCameraMatrix	:	TcVnMatrix3x3_LREAL;	(* Camera matrix containing the intrinsic parameters *)
		aDistortionCoefficients	:	TcVnArray8_LREAL;	(* Lens distortion coefficients [k1, k2, p1, p2, k3, k4, k5, k6] *)
		aNewCameraMatrix	:	TcVnMatrix3x3_LREAL;	(* Allows additional scaling and shifting of the result image *)
	END_VAR
	VAR_INPUT
		hrPrev	:	HRESULT;	(* HRESULT indicating the result of previous operations (If SUCCEEDED(hrPrev) equals false, no operation is executed.) *)
	END_VAR

END_FUNCTION

// Functions/Geometric and Coordinate Transformations/Calibration/F_VN_CompensateLensDistortionForPoints

	{attribute 'TcIecLibraryType'}
	{attribute 'external_name' := 'F_VN_CompensateLensDistortionForPoints_GUID_F502477C_D1E5_4E07_C519_51B41882E35B'}
	(* Transforms point coordinates to compensate the lens distortion. *)
	FUNCTION F_VN_CompensateLensDistortionForPoints : HRESULT
	VAR_INPUT
		ipSrcPoints	:	ITcVnContainer;	(* Container with source point coordinates (ContainerType_Vector_TcVnPoint2_REAL or ContainerType_Vector_TcVnPoint2_DINT) *)
		ipDestPoints	:	REFERENCE TO ITcVnContainer;	(* Returns a container with the transformed point coordinates (ContainerType_Vector_TcVnPoint2_REAL) *)
	END_VAR
	VAR_IN_OUT
		aCameraMatrix	:	TcVnMatrix3x3_LREAL;	(* Camera matrix containing the intrinsic parameters *)
		aDistortionCoefficients	:	TcVnArray4_LREAL;	(* Lens distortion coefficients [k1, k2, p1, p2] *)
	END_VAR
	VAR_INPUT
		hrPrev	:	HRESULT;	(* HRESULT indicating the result of previous operations (If SUCCEEDED(hrPrev) equals false, no operation is executed.) *)
	END_VAR

END_FUNCTION

// Functions/Geometric and Coordinate Transformations/Calibration/F_VN_CompensateLensDistortionForPointsExp1

	{attribute 'TcIecLibraryType'}
	{attribute 'external_name' := 'F_VN_CompensateLensDistortionForPointsExp1_GUID_94F790C8_D2D2_4E2F_F43B_7E2DC19348D5'}
	(* Transforms point coordinates to compensate the lens distortion. (expert function) *)
	FUNCTION F_VN_CompensateLensDistortionForPointsExp1 : HRESULT
	VAR_INPUT
		ipSrcPoints	:	ITcVnContainer;	(* Container with source point coordinates (ContainerType_Vector_TcVnPoint2_REAL or ContainerType_Vector_TcVnPoint2_DINT) *)
		ipDestPoints	:	REFERENCE TO ITcVnContainer;	(* Returns a container with the transformed point coordinates (ContainerType_Vector_TcVnPoint2_REAL) *)
	END_VAR
	VAR_IN_OUT
		aCameraMatrix	:	TcVnMatrix3x3_LREAL;	(* Camera matrix containing the intrinsic parameters *)
		aDistortionCoefficients	:	TcVnArray8_LREAL;	(* Lens distortion coefficients [k1, k2, p1, p2, k3, k4, k5, k6] *)
	END_VAR
	VAR_INPUT
		hrPrev	:	HRESULT;	(* HRESULT indicating the result of previous operations (If SUCCEEDED(hrPrev) equals false, no operation is executed.) *)
	END_VAR

END_FUNCTION

// Functions/Geometric and Coordinate Transformations/Calibration/F_VN_CompensateLensDistortionForPointsExp2

	{attribute 'TcIecLibraryType'}
	{attribute 'external_name' := 'F_VN_CompensateLensDistortionForPointsExp2_GUID_DB26C427_67A5_441B_D6BF_F08B21BCB900'}
	(* Transforms point coordinates to compensate the lens distortion. (expert function) *)
	FUNCTION F_VN_CompensateLensDistortionForPointsExp2 : HRESULT
	VAR_INPUT
		ipSrcPoints	:	ITcVnContainer;	(* Container with source point coordinates (ContainerType_Vector_TcVnPoint2_REAL or ContainerType_Vector_TcVnPoint2_DINT) *)
		ipDestPoints	:	REFERENCE TO ITcVnContainer;	(* Returns a container with the transformed point coordinates (ContainerType_Vector_TcVnPoint2_REAL) *)
	END_VAR
	VAR_IN_OUT
		aCameraMatrix	:	TcVnMatrix3x3_LREAL;	(* Camera matrix containing the intrinsic parameters *)
		aDistortionCoefficients	:	TcVnArray8_LREAL;	(* Lens distortion coefficients [k1, k2, p1, p2, k3, k4, k5, k6] *)
		aNewCameraMatrix	:	TcVnMatrix3x3_LREAL;	(* Allows additional shifting of the result point coordinates *)
	END_VAR
	VAR_INPUT
		hrPrev	:	HRESULT;	(* HRESULT indicating the result of previous operations (If SUCCEEDED(hrPrev) equals false, no operation is executed.) *)
	END_VAR

END_FUNCTION

// Functions/Geometric and Coordinate Transformations/Calibration/F_VN_DetectPatternPoints

	{attribute 'TcIecLibraryType'}
	{attribute 'external_name' := 'F_VN_DetectPatternPoints_GUID_0EC9B0C1_0375_48BD_DAC8_ED2738DD1537'}
	(* Detects calibration pattern points (circles) within the provided image. *)
	FUNCTION F_VN_DetectPatternPoints : HRESULT
	VAR_INPUT
		ipSrcImage	:	ITcVnImage;	(* Source image (USINT, 1 channel) *)
		ipPatternPoints	:	REFERENCE TO ITcVnContainer;	(* Returns the pattern point positions (ContainerType_Vector_TcVnPoint2_REAL; Non-zero interface pointers are reused.) *)
	END_VAR
	VAR_IN_OUT
		stBlobDetectionParams	:	TcVnParamsBlobDetection;	(* Parameters to detect and filter contours. *)
	END_VAR
	VAR_INPUT
		nNumberOfPoints	:	UDINT;	(* Expected number of pattern points *)
		hrPrev	:	HRESULT;	(* HRESULT indicating the result of previous operations (If SUCCEEDED(hrPrev) equals false, no operation is executed.) *)
	END_VAR

END_FUNCTION

// Functions/Geometric and Coordinate Transformations/Calibration/F_VN_DetectPatternPointsExp

	{attribute 'TcIecLibraryType'}
	{attribute 'external_name' := 'F_VN_DetectPatternPointsExp_GUID_E0A6CB71_643B_46EC_CD01_F55B68A730DF'}
	(* Detects calibration pattern points (circles) within the provided image. (expert function) *)
	FUNCTION F_VN_DetectPatternPointsExp : HRESULT
	VAR_INPUT
		ipSrcImage	:	ITcVnImage;	(* Source image (USINT, 1 channel) *)
		ipPatternPoints	:	REFERENCE TO ITcVnContainer;	(* Returns the pattern point positions (ContainerType_Vector_TcVnPoint2_REAL; Non-zero interface pointers are reused.) *)
	END_VAR
	VAR_IN_OUT
		stBlobDetectionParams	:	TcVnParamsBlobDetection;	(* Parameters to detect and filter contours. *)
	END_VAR
	VAR_INPUT
		nNumberOfPoints	:	UDINT;	(* Expected number of pattern points *)
		fSizeDiffThresFactor	:	REAL;	(* Threshold for filtering contours by average size *)
		bSubpixelAccuracy	:	BOOL;	(* If true, the pattern points are detected with subpixel accuracy *)
		eEdgeDirection	:	ETcVnEdgeDirection;	(* Specification of the edge direction to search for (from center to outside circle) *)
		fMinStrength	:	REAL;	(* Specification of the minimum strength (intensity difference) of the edge to search for *)
		nMaxThickness	:	UDINT;	(* Specification of the maximum thickness of the edge to search for, which means fMinStrength must be reached within nMaxThickness pixels *)
		nSubpixelsIterations	:	UDINT;	(* Specifies the number of subpixels (for INTERPOLATION, 10 - 20 usually is sufficient) or maximum number of iterations for optimizing the parameters (for APPROX_ERF and APPROX_GAUSSIAN, 50 - 100 usually is sufficient) *)
		nSearchLines	:	UDINT;	(* Specifies the amount of search lines, which are equally distributed in all directions (must be >= 8 and a multiple of 4) *)
		fApproxPrecision	:	REAL;	(* Specifies the approximation precision for APPROX_ERF and APPROX_GAUSSIAN (0.001 usually is sufficient, unused for INTERPOLATION) *)
		eAlgorithm	:	ETcVnEdgeDetectionAlgorithm;	(* Selection of the edge detection algorithm *)
		hrPrev	:	HRESULT;	(* HRESULT indicating the result of previous operations (If SUCCEEDED(hrPrev) equals false, no operation is executed.) *)
	END_VAR

END_FUNCTION

// Functions/Geometric and Coordinate Transformations/Calibration/F_VN_GenerateCalibrationPatternReferencePoints

	{attribute 'TcIecLibraryType'}
	{attribute 'external_name' := 'F_VN_GenerateCalibrationPatternReferencePoints_GUID_B6E9C829_B8C2_432B_D143_80CB7E3C1776'}
	(* Generate reference points for common calibration patterns. *)
	FUNCTION F_VN_GenerateCalibrationPatternReferencePoints : HRESULT
	VAR_INPUT
		ipReferencePoints	:	REFERENCE TO ITcVnContainer;	(* Returns the generated reference points (ContainerType_Vector_TcVnPoint3_REAL) *)
		ePattern	:	ETcVnCalibrationPattern;	(* Calibration pattern type *)
		eOrigin	:	ETcVnCalibrationPatternOrigin;	(* Calibration pattern origin *)
		nWidth	:	UDINT;	(* Pattern width, i.e. number of pattern points in x direction *)
		nHeight	:	UDINT;	(* Pattern height, i.e. number of pattern points in y direction *)
		fDistX	:	REAL;	(* Distance between pattern points in x direction *)
		fDistY	:	REAL;	(* Distance between pattern points in y direction *)
		hrPrev	:	HRESULT;	(* HRESULT indicating the result of previous operations (If SUCCEEDED(hrPrev) equals false, no operation is executed.) *)
	END_VAR

END_FUNCTION

// Functions/Geometric and Coordinate Transformations/Calibration/F_VN_ImagePointsWorldDistance

	{attribute 'TcIecLibraryType'}
	{attribute 'external_name' := 'F_VN_ImagePointsWorldDistance_GUID_E82B7700_985B_4FD9_E55E_24AE7140182D'}
	(* Computes the distance in the world coordinate system between two points (in the same world coordinate z layer) given in image coordinates. *)
	FUNCTION F_VN_ImagePointsWorldDistance : HRESULT
	VAR_IN_OUT
		aImagePoint1	:	TcVnPoint2_REAL;	(* First point in the image coordinate system *)
		aImagePoint2	:	TcVnPoint2_REAL;	(* Second point in the image coordinate system *)
		fWorldDistance	:	LREAL;	(* Returns the distance between aImagePoint1 and aImagePoint2 in the world coordinate system *)
		aCameraMatrix	:	TcVnMatrix3x3_LREAL;	(* 3x3 camera matrix containing the intrinsic parameters *)
		aDistortionCoefficients	:	TcVnArray8_LREAL;	(* Lens distortion coefficients [k1, k2, p1, p2, k3, k4, k5, k6] *)
		aRotationMatrix	:	TcVnMatrix3x3_LREAL;	(* 3x3 rotation matrix *)
		aTranslationVector	:	TcVnVector3_LREAL;	(* Translation vector *)
	END_VAR
	VAR_INPUT
		fZ	:	LREAL;	(* z coordinate (world coordinate system) of the given points (0 would be at (toplevel) calibration pattern) *)
		hrPrev	:	HRESULT;	(* HRESULT indicating the result of previous operations (If SUCCEEDED(hrPrev) equals false, no operation is executed.) *)
	END_VAR

END_FUNCTION

// Functions/Geometric and Coordinate Transformations/Calibration/F_VN_SolvePnP

	{attribute 'TcIecLibraryType'}
	{attribute 'external_name' := 'F_VN_SolvePnP_GUID_A3ADBE24_115D_419B_E35F_EB0C3BD18E9F'}
	(* Computes the rotation matrix and translation vector from 3D-2D point correspondences. *)
	FUNCTION F_VN_SolvePnP : HRESULT
	VAR_INPUT
		ipImagePoints	:	ITcVnContainer;	(* Image points (ContainerType_Vector_TcVnPoint2_REAL, requires at least 4 points in the same order as in ipReferencePoints) *)
		ipReferencePoints	:	ITcVnContainer;	(* Reference world points (ContainerType_Vector_TcVnPoint3_REAL, same number of points as in ipImagePoints) *)
	END_VAR
	VAR_IN_OUT
		aCameraMatrix	:	TcVnMatrix3x3_LREAL;	(* Camera matrix (e.g. computed with one of the CalibrateCamera functions) *)
		aDistortionCoefficients	:	TcVnArray8_LREAL;	(* Lens distortion coefficients [k1, k2, p1, p2, k3, k4, k5, k6] (e.g. computed with one of the CalibrateCamera functions) *)
		aRotationMatrix	:	TcVnMatrix3x3_LREAL;	(* Returns the rotation matrix *)
		aTranslationVector	:	TcVnVector3_LREAL;	(* Returns the translation vector *)
		fReprojError	:	LREAL;	(* Returns the reprojection error *)
	END_VAR
	VAR_INPUT
		hrPrev	:	HRESULT;	(* HRESULT indicating the result of previous operations (If SUCCEEDED(hrPrev) equals false, no operation is executed.) *)
	END_VAR

END_FUNCTION

// Functions/Geometric and Coordinate Transformations/Calibration/F_VN_SolvePnPExp

	{attribute 'TcIecLibraryType'}
	{attribute 'external_name' := 'F_VN_SolvePnPExp_GUID_A174FEDD_989C_43EC_CD41_EF9C6E280F18'}
	(* Computes the rotation matrix and translation vector from 3D-2D point correspondences. (expert function) *)
	FUNCTION F_VN_SolvePnPExp : HRESULT
	VAR_INPUT
		ipImagePoints	:	ITcVnContainer;	(* Image points (ContainerType_Vector_TcVnPoint2_REAL, requires at least 4 points in the same order as in ipReferencePoints) *)
		ipReferencePoints	:	ITcVnContainer;	(* Reference world points (ContainerType_Vector_TcVnPoint3_REAL, same number of points as in ipImagePoints) *)
	END_VAR
	VAR_IN_OUT
		aCameraMatrix	:	TcVnMatrix3x3_LREAL;	(* Camera matrix (e.g. computed with one of the CalibrateCamera functions) *)
		aDistortionCoefficients	:	TcVnArray8_LREAL;	(* Lens distortion coefficients [k1, k2, p1, p2, k3, k4, k5, k6] (e.g. computed with one of the CalibrateCamera functions) *)
		aRotationMatrix	:	TcVnMatrix3x3_LREAL;	(* Returns the rotation matrix *)
		aTranslationVector	:	TcVnVector3_LREAL;	(* Returns the translation vector *)
		fReprojError	:	LREAL;	(* Returns the reprojection error *)
	END_VAR
	VAR_INPUT
		eMethod	:	ETcVnSolvePnPMethod;	(* Solve PnP method *)
		bUseExtrinsicGuess	:	BOOL;	(* If true, the provided rotation matrix and translation vector are used as an initial guess for further optimization (only supported for the SPM_ITERATIVE method). *)
		hrPrev	:	HRESULT;	(* HRESULT indicating the result of previous operations (If SUCCEEDED(hrPrev) equals false, no operation is executed.) *)
	END_VAR

END_FUNCTION

// Functions/Geometric and Coordinate Transformations/Calibration/F_VN_SortDetectedPatternPoints

	{attribute 'TcIecLibraryType'}
	{attribute 'external_name' := 'F_VN_SortDetectedPatternPoints_GUID_4A60C343_CDC5_4055_C8B0_C2A46B82500C'}
	(* Sort the detected pattern points according to the relative positions of the calibration pattern points. *)
	FUNCTION F_VN_SortDetectedPatternPoints : HRESULT
	VAR_INPUT
		ipImagePoints	:	ITcVnContainer;	(* Detected pattern point positions in the image coordinate system (will be sorted by this function, ContainerType_Vector_TcVnPoint2_REAL) *)
		ipPatternPoints	:	ITcVnContainer;	(* The pattern points in the calibration pattern coordinate system, used as a reference to sort ipImagePoints (ContainerType_Vector_TcVnPoint3_REAL) *)
		hrPrev	:	HRESULT;	(* HRESULT indicating the result of previous operations (If SUCCEEDED(hrPrev) equals false, no operation is executed.) *)
	END_VAR

END_FUNCTION

// Functions/Geometric and Coordinate Transformations/Calibration/F_VN_TransformCoordinatesPlanar_Container

	{attribute 'TcIecLibraryType'}
	{attribute 'external_name' := 'F_VN_TransformCoordinatesPlanar_Container_GUID_8827D582_B0A5_4556_E512_120CF30D8594'}
	(* Compute real-world coordinates for given image points or vice versa. *)
	FUNCTION F_VN_TransformCoordinatesPlanar_Container : HRESULT
	VAR_INPUT
		ipSrcPoints	:	ITcVnContainer;	(* Container with 2D source points (TcVnPoint2_DINT or TcVnPoint2_REAL or TcVnPoint2_LREAL) *)
		ipDestPoints	:	REFERENCE TO ITcVnContainer;	(* Returns the transformed 2D points (TcVnPoint2_LREAL) *)
	END_VAR
	VAR_IN_OUT
		aTransformationMatrix	:	TcVnMatrix3x3_LREAL;	(* Transformation matrix obtained with VnCalibrateCameraPlanar() or its inverse matrix obtained with VnInvertMatrix3x3() *)
	END_VAR
	VAR_INPUT
		hrPrev	:	HRESULT;	(* HRESULT indicating the result of previous operations (If SUCCEEDED(hrPrev) equals false, no operation is executed.) *)
	END_VAR

END_FUNCTION

// Functions/Geometric and Coordinate Transformations/Calibration/F_VN_TransformCoordinatesPlanar_Point

	{attribute 'TcIecLibraryType'}
	{attribute 'external_name' := 'F_VN_TransformCoordinatesPlanar_Point_GUID_7CDD689E_9F56_46BC_EBCE_C39EC752046E'}
	(* Compute real-world coordinates for a given image point or vice versa. *)
	FUNCTION F_VN_TransformCoordinatesPlanar_Point : HRESULT
	VAR_IN_OUT
		aSrcPoint	:	TcVnPoint2_LREAL;	(* Point in the source coordinate system *)
		aDestPoint	:	TcVnPoint2_LREAL;	(* Returns point in the destination coordinate system *)
		aTransformationMatrix	:	TcVnMatrix3x3_LREAL;	(* Transformation matrix obtained with VnCalibrateCameraPlanar() or its inverse matrix obtained with VnInvertMatrix3x3() *)
	END_VAR
	VAR_INPUT
		hrPrev	:	HRESULT;	(* HRESULT indicating the result of previous operations (If SUCCEEDED(hrPrev) equals false, no operation is executed.) *)
	END_VAR

END_FUNCTION

// Functions/Geometric and Coordinate Transformations/Calibration/F_VN_TransformCoordinatesImageToWorld_Container

	{attribute 'TcIecLibraryType'}
	{attribute 'external_name' := 'F_VN_TransformCoordinatesImageToWorld_Container_GUID_BBB07077_C4D3_44F3_DA38_DA590AF477DE'}
	(* Transform 2D image point coordinates to 3D world coordinates (using intrinsic + extrinsic calibration results). *)
	FUNCTION F_VN_TransformCoordinatesImageToWorld_Container : HRESULT
	VAR_INPUT
		ipSrcPoints2D	:	ITcVnContainer;	(* Container with 2D source points (TcVnPoint2_DINT or TcVnPoint2_REAL or TcVnPoint2_LREAL) *)
		ipDestPoints3D	:	REFERENCE TO ITcVnContainer;	(* Returns the transformed 3D points (TcVnPoint3_LREAL) *)
	END_VAR
	VAR_IN_OUT
		aCameraMatrix	:	TcVnMatrix3x3_LREAL;	(* 3x3 camera matrix containing the intrinsic parameters *)
		aDistortionCoefficients	:	TcVnArray8_LREAL;	(* Lens distortion coefficients [k1, k2, p1, p2, k3, k4, k5, k6] *)
		aRotationMatrix	:	TcVnMatrix3x3_LREAL;	(* 3x3 rotation matrix *)
		aTranslationVector	:	TcVnVector3_LREAL;	(* Translation vector *)
	END_VAR
	VAR_INPUT
		fZ	:	LREAL;	(* z coordinate (world coordinate system) of the transformed points (0 would be at (toplevel) calibration pattern) *)
		hrPrev	:	HRESULT;	(* HRESULT indicating the result of previous operations (If SUCCEEDED(hrPrev) equals false, no operation is executed.) *)
	END_VAR

END_FUNCTION

// Functions/Geometric and Coordinate Transformations/Calibration/F_VN_TransformCoordinatesImageToWorld_Point

	{attribute 'TcIecLibraryType'}
	{attribute 'external_name' := 'F_VN_TransformCoordinatesImageToWorld_Point_GUID_6C929981_F020_4537_ECD5_CBCD852A1A80'}
	(* Transform 2D image point coordinate to 3D world coordinate (using intrinsic + extrinsic calibration results). *)
	FUNCTION F_VN_TransformCoordinatesImageToWorld_Point : HRESULT
	VAR_IN_OUT
		aSrcPoint	:	TcVnPoint2_LREAL;	(* Point in the image coordinate system *)
		aDestPoint	:	TcVnPoint3_LREAL;	(* Returns the point in the world coordinate system *)
		aCameraMatrix	:	TcVnMatrix3x3_LREAL;	(* 3x3 camera matrix containing the intrinsic parameters *)
		aDistortionCoefficients	:	TcVnArray8_LREAL;	(* Lens distortion coefficients [k1, k2, p1, p2, k3, k4, k5, k6] *)
		aRotationMatrix	:	TcVnMatrix3x3_LREAL;	(* 3x3 rotation matrix *)
		aTranslationVector	:	TcVnVector3_LREAL;	(* Translation vector *)
	END_VAR
	VAR_INPUT
		fZ	:	LREAL;	(* z coordinate (world coordinate system) of the transformed points (0 would be at (toplevel) calibration pattern) *)
		hrPrev	:	HRESULT;	(* HRESULT indicating the result of previous operations (If SUCCEEDED(hrPrev) equals false, no operation is executed.) *)
	END_VAR

END_FUNCTION

// Functions/Geometric and Coordinate Transformations/Calibration/F_VN_TransformCoordinatesWorldToImage_Container

	{attribute 'TcIecLibraryType'}
	{attribute 'external_name' := 'F_VN_TransformCoordinatesWorldToImage_Container_GUID_29A66D73_DFD3_4B7F_EC44_6564B5859BFE'}
	(* Transform 3D world coordinates to 2D image coordinates (using intrinsic + extrinsic calibration results). *)
	FUNCTION F_VN_TransformCoordinatesWorldToImage_Container : HRESULT
	VAR_INPUT
		ipSrcPoints3D	:	ITcVnContainer;	(* Container with 3D source points (TcVnPoint3_LREAL) *)
		ipDestPoints2D	:	REFERENCE TO ITcVnContainer;	(* Returns the transformed 2D points (TcVnPoint2_REAL or TcVnPoint2_DINT, depending on bInteger) *)
	END_VAR
	VAR_IN_OUT
		aCameraMatrix	:	TcVnMatrix3x3_LREAL;	(* 3x3 camera matrix containing the intrinsic parameters *)
		aDistortionCoefficients	:	TcVnArray8_LREAL;	(* Lens distortion coefficients [k1, k2, p1, p2, k3, k4, k5, k6] *)
		aRotationMatrix	:	TcVnMatrix3x3_LREAL;	(* 3x3 rotation matrix *)
		aTranslationVector	:	TcVnVector3_LREAL;	(* Translation vector *)
	END_VAR
	VAR_INPUT
		bInteger	:	BOOL;	(* Selects whether the function returns a container of TcVnPoint2_DINT or TcVnPoint2_REAL *)
		hrPrev	:	HRESULT;	(* HRESULT indicating the result of previous operations (If SUCCEEDED(hrPrev) equals false, no operation is executed.) *)
	END_VAR

END_FUNCTION

// Functions/Geometric and Coordinate Transformations/Calibration/F_VN_TransformCoordinatesWorldToImage_Point

	{attribute 'TcIecLibraryType'}
	{attribute 'external_name' := 'F_VN_TransformCoordinatesWorldToImage_Point_GUID_6D940453_FC37_401D_EE1B_943AF5A61FF0'}
	(* Transform 3D world coordinates to 2D image coordinates (using intrinsic + extrinsic calibration results). *)
	FUNCTION F_VN_TransformCoordinatesWorldToImage_Point : HRESULT
	VAR_IN_OUT
		aSrcPoint	:	TcVnPoint3_LREAL;	(* 3D source point (world coordinate system) *)
		aDestPoint	:	TcVnPoint2_REAL;	(* Returns the transformed 2D point (image coordinate system) *)
		aCameraMatrix	:	TcVnMatrix3x3_LREAL;	(* 3x3 camera matrix containing the intrinsic parameters *)
		aDistortionCoefficients	:	TcVnArray8_LREAL;	(* Lens distortion coefficients [k1, k2, p1, p2, k3, k4, k5, k6] *)
		aRotationMatrix	:	TcVnMatrix3x3_LREAL;	(* 3x3 rotation matrix *)
		aTranslationVector	:	TcVnVector3_LREAL;	(* Translation vector *)
	END_VAR
	VAR_INPUT
		hrPrev	:	HRESULT;	(* HRESULT indicating the result of previous operations (If SUCCEEDED(hrPrev) equals false, no operation is executed.) *)
	END_VAR

END_FUNCTION

// Functions/Container Statistics/F_VN_MaxElementElementwise/F_VN_MaxElementElementwise_DINT

	{attribute 'TcIecLibraryType'}
	{attribute 'external_name' := 'F_VN_MaxElementElementwise_DINT_GUID_4AA1EB72_1242_4EF2_D489_899C7CCB6856'}
	(* Gets the element wise maximum container element. *)
	FUNCTION F_VN_MaxElementElementwise_DINT : HRESULT
	VAR_INPUT
		ipContainer	:	ITcVnContainer;	(* Source container *)
	END_VAR
	VAR_IN_OUT
		nMax	:	DINT;	(* Returns the requested element *)
	END_VAR
	VAR_INPUT
		hrPrev	:	HRESULT;	(* HRESULT indicating the result of previous operations (If SUCCEEDED(hrPrev) equals false, no operation is executed.) *)
	END_VAR

END_FUNCTION

// Functions/Container Statistics/F_VN_MaxElementElementwise/F_VN_MaxElementElementwise_INT

	{attribute 'TcIecLibraryType'}
	{attribute 'external_name' := 'F_VN_MaxElementElementwise_INT_GUID_7EA866C5_A781_4D59_EF6C_C96445691A86'}
	(* Gets the element wise maximum container element. *)
	FUNCTION F_VN_MaxElementElementwise_INT : HRESULT
	VAR_INPUT
		ipContainer	:	ITcVnContainer;	(* Source container *)
	END_VAR
	VAR_IN_OUT
		nMax	:	INT;	(* Returns the requested element *)
	END_VAR
	VAR_INPUT
		hrPrev	:	HRESULT;	(* HRESULT indicating the result of previous operations (If SUCCEEDED(hrPrev) equals false, no operation is executed.) *)
	END_VAR

END_FUNCTION

// Functions/Container Statistics/F_VN_MaxElementElementwise/F_VN_MaxElementElementwise_LREAL

	{attribute 'TcIecLibraryType'}
	{attribute 'external_name' := 'F_VN_MaxElementElementwise_LREAL_GUID_A9159211_B5A6_419E_EEFF_082BEB61B8F8'}
	(* Gets the element wise maximum container element. *)
	FUNCTION F_VN_MaxElementElementwise_LREAL : HRESULT
	VAR_INPUT
		ipContainer	:	ITcVnContainer;	(* Source container *)
	END_VAR
	VAR_IN_OUT
		fMax	:	LREAL;	(* Returns the requested element *)
	END_VAR
	VAR_INPUT
		hrPrev	:	HRESULT;	(* HRESULT indicating the result of previous operations (If SUCCEEDED(hrPrev) equals false, no operation is executed.) *)
	END_VAR

END_FUNCTION

// Functions/Container Statistics/F_VN_MaxElementElementwise/F_VN_MaxElementElementwise_REAL

	{attribute 'TcIecLibraryType'}
	{attribute 'external_name' := 'F_VN_MaxElementElementwise_REAL_GUID_C2E426E4_21C7_4CBD_E3FF_E3986A4C6276'}
	(* Gets the element wise maximum container element. *)
	FUNCTION F_VN_MaxElementElementwise_REAL : HRESULT
	VAR_INPUT
		ipContainer	:	ITcVnContainer;	(* Source container *)
	END_VAR
	VAR_IN_OUT
		fMax	:	REAL;	(* Returns the requested element *)
	END_VAR
	VAR_INPUT
		hrPrev	:	HRESULT;	(* HRESULT indicating the result of previous operations (If SUCCEEDED(hrPrev) equals false, no operation is executed.) *)
	END_VAR

END_FUNCTION

// Functions/Container Statistics/F_VN_MaxElementElementwise/F_VN_MaxElementElementwise_SINT

	{attribute 'TcIecLibraryType'}
	{attribute 'external_name' := 'F_VN_MaxElementElementwise_SINT_GUID_3C750DB1_FDF5_43B1_C4DC_AE14EDE1538C'}
	(* Gets the element wise maximum container element. *)
	FUNCTION F_VN_MaxElementElementwise_SINT : HRESULT
	VAR_INPUT
		ipContainer	:	ITcVnContainer;	(* Source container *)
	END_VAR
	VAR_IN_OUT
		nMax	:	SINT;	(* Returns the requested element *)
	END_VAR
	VAR_INPUT
		hrPrev	:	HRESULT;	(* HRESULT indicating the result of previous operations (If SUCCEEDED(hrPrev) equals false, no operation is executed.) *)
	END_VAR

END_FUNCTION

// Functions/Container Statistics/F_VN_MaxElementElementwise/F_VN_MaxElementElementwise_TcVnPoint2_DINT

	{attribute 'TcIecLibraryType'}
	{attribute 'external_name' := 'F_VN_MaxElementElementwise_TcVnPoint2_DINT_GUID_4092E1EB_3605_4FB3_F6DA_41B6278A6555'}
	(* Gets the element wise maximum container element. *)
	FUNCTION F_VN_MaxElementElementwise_TcVnPoint2_DINT : HRESULT
	VAR_INPUT
		ipContainer	:	ITcVnContainer;	(* Source container *)
	END_VAR
	VAR_IN_OUT
		aMax	:	TcVnPoint2_DINT;	(* Returns the requested element *)
	END_VAR
	VAR_INPUT
		hrPrev	:	HRESULT;	(* HRESULT indicating the result of previous operations (If SUCCEEDED(hrPrev) equals false, no operation is executed.) *)
	END_VAR

END_FUNCTION

// Functions/Container Statistics/F_VN_MaxElementElementwise/F_VN_MaxElementElementwise_TcVnPoint2_LREAL

	{attribute 'TcIecLibraryType'}
	{attribute 'external_name' := 'F_VN_MaxElementElementwise_TcVnPoint2_LREAL_GUID_4EF2ACC7_7AC6_4F22_D3AC_E702C294E0E5'}
	(* Gets the element wise maximum container element. *)
	FUNCTION F_VN_MaxElementElementwise_TcVnPoint2_LREAL : HRESULT
	VAR_INPUT
		ipContainer	:	ITcVnContainer;	(* Source container *)
	END_VAR
	VAR_IN_OUT
		aMax	:	TcVnPoint2_LREAL;	(* Returns the requested element *)
	END_VAR
	VAR_INPUT
		hrPrev	:	HRESULT;	(* HRESULT indicating the result of previous operations (If SUCCEEDED(hrPrev) equals false, no operation is executed.) *)
	END_VAR

END_FUNCTION

// Functions/Container Statistics/F_VN_MaxElementElementwise/F_VN_MaxElementElementwise_TcVnPoint2_REAL

	{attribute 'TcIecLibraryType'}
	{attribute 'external_name' := 'F_VN_MaxElementElementwise_TcVnPoint2_REAL_GUID_E50BAEC1_ADB8_4C46_F126_84D05F09AC71'}
	(* Gets the element wise maximum container element. *)
	FUNCTION F_VN_MaxElementElementwise_TcVnPoint2_REAL : HRESULT
	VAR_INPUT
		ipContainer	:	ITcVnContainer;	(* Source container *)
	END_VAR
	VAR_IN_OUT
		aMax	:	TcVnPoint2_REAL;	(* Returns the requested element *)
	END_VAR
	VAR_INPUT
		hrPrev	:	HRESULT;	(* HRESULT indicating the result of previous operations (If SUCCEEDED(hrPrev) equals false, no operation is executed.) *)
	END_VAR

END_FUNCTION

// Functions/Container Statistics/F_VN_MaxElementElementwise/F_VN_MaxElementElementwise_TcVnPoint3_LREAL

	{attribute 'TcIecLibraryType'}
	{attribute 'external_name' := 'F_VN_MaxElementElementwise_TcVnPoint3_LREAL_GUID_E15ECB19_1B77_425B_D266_77AD3E920AD7'}
	(* Gets the element wise maximum container element. *)
	FUNCTION F_VN_MaxElementElementwise_TcVnPoint3_LREAL : HRESULT
	VAR_INPUT
		ipContainer	:	ITcVnContainer;	(* Source container *)
	END_VAR
	VAR_IN_OUT
		aMax	:	TcVnPoint3_LREAL;	(* Returns the requested element *)
	END_VAR
	VAR_INPUT
		hrPrev	:	HRESULT;	(* HRESULT indicating the result of previous operations (If SUCCEEDED(hrPrev) equals false, no operation is executed.) *)
	END_VAR

END_FUNCTION

// Functions/Container Statistics/F_VN_MaxElementElementwise/F_VN_MaxElementElementwise_TcVnPoint3_REAL

	{attribute 'TcIecLibraryType'}
	{attribute 'external_name' := 'F_VN_MaxElementElementwise_TcVnPoint3_REAL_GUID_1683DCEB_8C71_43F7_D54D_57D3D7569B1A'}
	(* Gets the element wise maximum container element. *)
	FUNCTION F_VN_MaxElementElementwise_TcVnPoint3_REAL : HRESULT
	VAR_INPUT
		ipContainer	:	ITcVnContainer;	(* Source container *)
	END_VAR
	VAR_IN_OUT
		aMax	:	TcVnPoint3_REAL;	(* Returns the requested element *)
	END_VAR
	VAR_INPUT
		hrPrev	:	HRESULT;	(* HRESULT indicating the result of previous operations (If SUCCEEDED(hrPrev) equals false, no operation is executed.) *)
	END_VAR

END_FUNCTION

// Functions/Container Statistics/F_VN_MaxElementElementwise/F_VN_MaxElementElementwise_TcVnVector2_DINT

	{attribute 'TcIecLibraryType'}
	{attribute 'external_name' := 'F_VN_MaxElementElementwise_TcVnVector2_DINT_GUID_28FD57DA_E129_45BC_C5FA_AEB7497B749F'}
	(* Gets the element wise maximum container element. *)
	FUNCTION F_VN_MaxElementElementwise_TcVnVector2_DINT : HRESULT
	VAR_INPUT
		ipContainer	:	ITcVnContainer;	(* Source container *)
	END_VAR
	VAR_IN_OUT
		aMax	:	TcVnVector2_DINT;	(* Returns the requested element *)
	END_VAR
	VAR_INPUT
		hrPrev	:	HRESULT;	(* HRESULT indicating the result of previous operations (If SUCCEEDED(hrPrev) equals false, no operation is executed.) *)
	END_VAR

END_FUNCTION

// Functions/Container Statistics/F_VN_MaxElementElementwise/F_VN_MaxElementElementwise_TcVnVector2_INT

	{attribute 'TcIecLibraryType'}
	{attribute 'external_name' := 'F_VN_MaxElementElementwise_TcVnVector2_INT_GUID_21721B2E_B70F_4F31_D976_2FBDD21CCF0F'}
	(* Gets the element wise maximum container element. *)
	FUNCTION F_VN_MaxElementElementwise_TcVnVector2_INT : HRESULT
	VAR_INPUT
		ipContainer	:	ITcVnContainer;	(* Source container *)
	END_VAR
	VAR_IN_OUT
		aMax	:	TcVnVector2_INT;	(* Returns the requested element *)
	END_VAR
	VAR_INPUT
		hrPrev	:	HRESULT;	(* HRESULT indicating the result of previous operations (If SUCCEEDED(hrPrev) equals false, no operation is executed.) *)
	END_VAR

END_FUNCTION

// Functions/Container Statistics/F_VN_MaxElementElementwise/F_VN_MaxElementElementwise_TcVnVector2_REAL

	{attribute 'TcIecLibraryType'}
	{attribute 'external_name' := 'F_VN_MaxElementElementwise_TcVnVector2_REAL_GUID_466178CC_049F_497A_C56B_F7B37766D164'}
	(* Gets the element wise maximum container element. *)
	FUNCTION F_VN_MaxElementElementwise_TcVnVector2_REAL : HRESULT
	VAR_INPUT
		ipContainer	:	ITcVnContainer;	(* Source container *)
	END_VAR
	VAR_IN_OUT
		aMax	:	TcVnVector2_REAL;	(* Returns the requested element *)
	END_VAR
	VAR_INPUT
		hrPrev	:	HRESULT;	(* HRESULT indicating the result of previous operations (If SUCCEEDED(hrPrev) equals false, no operation is executed.) *)
	END_VAR

END_FUNCTION

// Functions/Container Statistics/F_VN_MaxElementElementwise/F_VN_MaxElementElementwise_TcVnVector2_SINT

	{attribute 'TcIecLibraryType'}
	{attribute 'external_name' := 'F_VN_MaxElementElementwise_TcVnVector2_SINT_GUID_C2BCC6D6_720F_4410_E32F_CBAEF8149DA7'}
	(* Gets the element wise maximum container element. *)
	FUNCTION F_VN_MaxElementElementwise_TcVnVector2_SINT : HRESULT
	VAR_INPUT
		ipContainer	:	ITcVnContainer;	(* Source container *)
	END_VAR
	VAR_IN_OUT
		aMax	:	TcVnVector2_SINT;	(* Returns the requested element *)
	END_VAR
	VAR_INPUT
		hrPrev	:	HRESULT;	(* HRESULT indicating the result of previous operations (If SUCCEEDED(hrPrev) equals false, no operation is executed.) *)
	END_VAR

END_FUNCTION

// Functions/Container Statistics/F_VN_MaxElementElementwise/F_VN_MaxElementElementwise_TcVnVector2_UINT

	{attribute 'TcIecLibraryType'}
	{attribute 'external_name' := 'F_VN_MaxElementElementwise_TcVnVector2_UINT_GUID_50612518_DF3D_4E3E_E2DB_DDF7BEE88DA3'}
	(* Gets the element wise maximum container element. *)
	FUNCTION F_VN_MaxElementElementwise_TcVnVector2_UINT : HRESULT
	VAR_INPUT
		ipContainer	:	ITcVnContainer;	(* Source container *)
	END_VAR
	VAR_IN_OUT
		aMax	:	TcVnVector2_UINT;	(* Returns the requested element *)
	END_VAR
	VAR_INPUT
		hrPrev	:	HRESULT;	(* HRESULT indicating the result of previous operations (If SUCCEEDED(hrPrev) equals false, no operation is executed.) *)
	END_VAR

END_FUNCTION

// Functions/Container Statistics/F_VN_MaxElementElementwise/F_VN_MaxElementElementwise_TcVnVector2_USINT

	{attribute 'TcIecLibraryType'}
	{attribute 'external_name' := 'F_VN_MaxElementElementwise_TcVnVector2_USINT_GUID_0509ED59_5506_4819_E3ED_418779A39CCE'}
	(* Gets the element wise maximum container element. *)
	FUNCTION F_VN_MaxElementElementwise_TcVnVector2_USINT : HRESULT
	VAR_INPUT
		ipContainer	:	ITcVnContainer;	(* Source container *)
	END_VAR
	VAR_IN_OUT
		aMax	:	TcVnVector2_USINT;	(* Returns the requested element *)
	END_VAR
	VAR_INPUT
		hrPrev	:	HRESULT;	(* HRESULT indicating the result of previous operations (If SUCCEEDED(hrPrev) equals false, no operation is executed.) *)
	END_VAR

END_FUNCTION

// Functions/Container Statistics/F_VN_MaxElementElementwise/F_VN_MaxElementElementwise_TcVnVector3_INT

	{attribute 'TcIecLibraryType'}
	{attribute 'external_name' := 'F_VN_MaxElementElementwise_TcVnVector3_INT_GUID_F29F56C7_86F6_4412_FDE1_5D89CB2266A8'}
	(* Gets the element wise maximum container element. *)
	FUNCTION F_VN_MaxElementElementwise_TcVnVector3_INT : HRESULT
	VAR_INPUT
		ipContainer	:	ITcVnContainer;	(* Source container *)
	END_VAR
	VAR_IN_OUT
		aMax	:	TcVnVector3_INT;	(* Returns the requested element *)
	END_VAR
	VAR_INPUT
		hrPrev	:	HRESULT;	(* HRESULT indicating the result of previous operations (If SUCCEEDED(hrPrev) equals false, no operation is executed.) *)
	END_VAR

END_FUNCTION

// Functions/Container Statistics/F_VN_MaxElementElementwise/F_VN_MaxElementElementwise_TcVnVector3_REAL

	{attribute 'TcIecLibraryType'}
	{attribute 'external_name' := 'F_VN_MaxElementElementwise_TcVnVector3_REAL_GUID_7129AC26_24A1_481E_F685_8FF54CAD9CF4'}
	(* Gets the element wise maximum container element. *)
	FUNCTION F_VN_MaxElementElementwise_TcVnVector3_REAL : HRESULT
	VAR_INPUT
		ipContainer	:	ITcVnContainer;	(* Source container *)
	END_VAR
	VAR_IN_OUT
		aMax	:	TcVnVector3_REAL;	(* Returns the requested element *)
	END_VAR
	VAR_INPUT
		hrPrev	:	HRESULT;	(* HRESULT indicating the result of previous operations (If SUCCEEDED(hrPrev) equals false, no operation is executed.) *)
	END_VAR

END_FUNCTION

// Functions/Container Statistics/F_VN_MaxElementElementwise/F_VN_MaxElementElementwise_TcVnVector3_SINT

	{attribute 'TcIecLibraryType'}
	{attribute 'external_name' := 'F_VN_MaxElementElementwise_TcVnVector3_SINT_GUID_12624EF9_375E_4917_E282_9ACC3C8A25B2'}
	(* Gets the element wise maximum container element. *)
	FUNCTION F_VN_MaxElementElementwise_TcVnVector3_SINT : HRESULT
	VAR_INPUT
		ipContainer	:	ITcVnContainer;	(* Source container *)
	END_VAR
	VAR_IN_OUT
		aMax	:	TcVnVector3_SINT;	(* Returns the requested element *)
	END_VAR
	VAR_INPUT
		hrPrev	:	HRESULT;	(* HRESULT indicating the result of previous operations (If SUCCEEDED(hrPrev) equals false, no operation is executed.) *)
	END_VAR

END_FUNCTION

// Functions/Container Statistics/F_VN_MaxElementElementwise/F_VN_MaxElementElementwise_TcVnVector3_UINT

	{attribute 'TcIecLibraryType'}
	{attribute 'external_name' := 'F_VN_MaxElementElementwise_TcVnVector3_UINT_GUID_6754DD0A_2E0B_442D_CD6B_2B5008F399CE'}
	(* Gets the element wise maximum container element. *)
	FUNCTION F_VN_MaxElementElementwise_TcVnVector3_UINT : HRESULT
	VAR_INPUT
		ipContainer	:	ITcVnContainer;	(* Source container *)
	END_VAR
	VAR_IN_OUT
		aMax	:	TcVnVector3_UINT;	(* Returns the requested element *)
	END_VAR
	VAR_INPUT
		hrPrev	:	HRESULT;	(* HRESULT indicating the result of previous operations (If SUCCEEDED(hrPrev) equals false, no operation is executed.) *)
	END_VAR

END_FUNCTION

// Functions/Container Statistics/F_VN_MaxElementElementwise/F_VN_MaxElementElementwise_TcVnVector3_USINT

	{attribute 'TcIecLibraryType'}
	{attribute 'external_name' := 'F_VN_MaxElementElementwise_TcVnVector3_USINT_GUID_BAD421F0_421E_4AA6_FE05_7A6B0DD89499'}
	(* Gets the element wise maximum container element. *)
	FUNCTION F_VN_MaxElementElementwise_TcVnVector3_USINT : HRESULT
	VAR_INPUT
		ipContainer	:	ITcVnContainer;	(* Source container *)
	END_VAR
	VAR_IN_OUT
		aMax	:	TcVnVector3_USINT;	(* Returns the requested element *)
	END_VAR
	VAR_INPUT
		hrPrev	:	HRESULT;	(* HRESULT indicating the result of previous operations (If SUCCEEDED(hrPrev) equals false, no operation is executed.) *)
	END_VAR

END_FUNCTION

// Functions/Container Statistics/F_VN_MaxElementElementwise/F_VN_MaxElementElementwise_TcVnVector4_DINT

	{attribute 'TcIecLibraryType'}
	{attribute 'external_name' := 'F_VN_MaxElementElementwise_TcVnVector4_DINT_GUID_BDAC63D7_AAED_41C6_D895_2F4A1DC1DBBB'}
	(* Gets the element wise maximum container element. *)
	FUNCTION F_VN_MaxElementElementwise_TcVnVector4_DINT : HRESULT
	VAR_INPUT
		ipContainer	:	ITcVnContainer;	(* Source container *)
	END_VAR
	VAR_IN_OUT
		aMax	:	TcVnVector4_DINT;	(* Returns the requested element *)
	END_VAR
	VAR_INPUT
		hrPrev	:	HRESULT;	(* HRESULT indicating the result of previous operations (If SUCCEEDED(hrPrev) equals false, no operation is executed.) *)
	END_VAR

END_FUNCTION

// Functions/Container Statistics/F_VN_MaxElementElementwise/F_VN_MaxElementElementwise_TcVnVector4_INT

	{attribute 'TcIecLibraryType'}
	{attribute 'external_name' := 'F_VN_MaxElementElementwise_TcVnVector4_INT_GUID_6FB8AFA2_A45C_43C7_E657_8B8B36E39DF4'}
	(* Gets the element wise maximum container element. *)
	FUNCTION F_VN_MaxElementElementwise_TcVnVector4_INT : HRESULT
	VAR_INPUT
		ipContainer	:	ITcVnContainer;	(* Source container *)
	END_VAR
	VAR_IN_OUT
		aMax	:	TcVnVector4_INT;	(* Returns the requested element *)
	END_VAR
	VAR_INPUT
		hrPrev	:	HRESULT;	(* HRESULT indicating the result of previous operations (If SUCCEEDED(hrPrev) equals false, no operation is executed.) *)
	END_VAR

END_FUNCTION

// Functions/Container Statistics/F_VN_MaxElementElementwise/F_VN_MaxElementElementwise_TcVnVector4_LREAL

	{attribute 'TcIecLibraryType'}
	{attribute 'external_name' := 'F_VN_MaxElementElementwise_TcVnVector4_LREAL_GUID_879896CE_7D05_4ED9_EE4E_9CE6B2E6A3A0'}
	(* Gets the element wise maximum container element. *)
	FUNCTION F_VN_MaxElementElementwise_TcVnVector4_LREAL : HRESULT
	VAR_INPUT
		ipContainer	:	ITcVnContainer;	(* Source container *)
	END_VAR
	VAR_IN_OUT
		aMax	:	TcVnVector4_LREAL;	(* Returns the requested element *)
	END_VAR
	VAR_INPUT
		hrPrev	:	HRESULT;	(* HRESULT indicating the result of previous operations (If SUCCEEDED(hrPrev) equals false, no operation is executed.) *)
	END_VAR

END_FUNCTION

// Functions/Container Statistics/F_VN_MaxElementElementwise/F_VN_MaxElementElementwise_TcVnVector4_REAL

	{attribute 'TcIecLibraryType'}
	{attribute 'external_name' := 'F_VN_MaxElementElementwise_TcVnVector4_REAL_GUID_D72BB1A0_64A9_4259_D48E_3DB24DEAE85A'}
	(* Gets the element wise maximum container element. *)
	FUNCTION F_VN_MaxElementElementwise_TcVnVector4_REAL : HRESULT
	VAR_INPUT
		ipContainer	:	ITcVnContainer;	(* Source container *)
	END_VAR
	VAR_IN_OUT
		aMax	:	TcVnVector4_REAL;	(* Returns the requested element *)
	END_VAR
	VAR_INPUT
		hrPrev	:	HRESULT;	(* HRESULT indicating the result of previous operations (If SUCCEEDED(hrPrev) equals false, no operation is executed.) *)
	END_VAR

END_FUNCTION

// Functions/Container Statistics/F_VN_MaxElementElementwise/F_VN_MaxElementElementwise_TcVnVector4_SINT

	{attribute 'TcIecLibraryType'}
	{attribute 'external_name' := 'F_VN_MaxElementElementwise_TcVnVector4_SINT_GUID_CB296B4E_F12A_44C3_F91C_368FEA96EF85'}
	(* Gets the element wise maximum container element. *)
	FUNCTION F_VN_MaxElementElementwise_TcVnVector4_SINT : HRESULT
	VAR_INPUT
		ipContainer	:	ITcVnContainer;	(* Source container *)
	END_VAR
	VAR_IN_OUT
		aMax	:	TcVnVector4_SINT;	(* Returns the requested element *)
	END_VAR
	VAR_INPUT
		hrPrev	:	HRESULT;	(* HRESULT indicating the result of previous operations (If SUCCEEDED(hrPrev) equals false, no operation is executed.) *)
	END_VAR

END_FUNCTION

// Functions/Container Statistics/F_VN_MaxElementElementwise/F_VN_MaxElementElementwise_TcVnVector4_UINT

	{attribute 'TcIecLibraryType'}
	{attribute 'external_name' := 'F_VN_MaxElementElementwise_TcVnVector4_UINT_GUID_1573943E_DAC1_494D_E6AB_F88ADF31D94E'}
	(* Gets the element wise maximum container element. *)
	FUNCTION F_VN_MaxElementElementwise_TcVnVector4_UINT : HRESULT
	VAR_INPUT
		ipContainer	:	ITcVnContainer;	(* Source container *)
	END_VAR
	VAR_IN_OUT
		aMax	:	TcVnVector4_UINT;	(* Returns the requested element *)
	END_VAR
	VAR_INPUT
		hrPrev	:	HRESULT;	(* HRESULT indicating the result of previous operations (If SUCCEEDED(hrPrev) equals false, no operation is executed.) *)
	END_VAR

END_FUNCTION

// Functions/Container Statistics/F_VN_MaxElementElementwise/F_VN_MaxElementElementwise_TcVnVector4_USINT

	{attribute 'TcIecLibraryType'}
	{attribute 'external_name' := 'F_VN_MaxElementElementwise_TcVnVector4_USINT_GUID_ECAA4F04_0103_43BF_C78A_F81D4334EC51'}
	(* Gets the element wise maximum container element. *)
	FUNCTION F_VN_MaxElementElementwise_TcVnVector4_USINT : HRESULT
	VAR_INPUT
		ipContainer	:	ITcVnContainer;	(* Source container *)
	END_VAR
	VAR_IN_OUT
		aMax	:	TcVnVector4_USINT;	(* Returns the requested element *)
	END_VAR
	VAR_INPUT
		hrPrev	:	HRESULT;	(* HRESULT indicating the result of previous operations (If SUCCEEDED(hrPrev) equals false, no operation is executed.) *)
	END_VAR

END_FUNCTION

// Functions/Container Statistics/F_VN_MaxElementElementwise/F_VN_MaxElementElementwise_UDINT

	{attribute 'TcIecLibraryType'}
	{attribute 'external_name' := 'F_VN_MaxElementElementwise_UDINT_GUID_5FD56304_3AA6_4A0C_F5C7_951B49190896'}
	(* Gets the element wise maximum container element. *)
	FUNCTION F_VN_MaxElementElementwise_UDINT : HRESULT
	VAR_INPUT
		ipContainer	:	ITcVnContainer;	(* Source container *)
	END_VAR
	VAR_IN_OUT
		nMax	:	UDINT;	(* Returns the requested element *)
	END_VAR
	VAR_INPUT
		hrPrev	:	HRESULT;	(* HRESULT indicating the result of previous operations (If SUCCEEDED(hrPrev) equals false, no operation is executed.) *)
	END_VAR

END_FUNCTION

// Functions/Container Statistics/F_VN_MaxElementElementwise/F_VN_MaxElementElementwise_UINT

	{attribute 'TcIecLibraryType'}
	{attribute 'external_name' := 'F_VN_MaxElementElementwise_UINT_GUID_5C1BEB9B_1729_499A_D38E_6D333A3BB44D'}
	(* Gets the element wise maximum container element. *)
	FUNCTION F_VN_MaxElementElementwise_UINT : HRESULT
	VAR_INPUT
		ipContainer	:	ITcVnContainer;	(* Source container *)
	END_VAR
	VAR_IN_OUT
		nMax	:	UINT;	(* Returns the requested element *)
	END_VAR
	VAR_INPUT
		hrPrev	:	HRESULT;	(* HRESULT indicating the result of previous operations (If SUCCEEDED(hrPrev) equals false, no operation is executed.) *)
	END_VAR

END_FUNCTION

// Functions/Container Statistics/F_VN_MaxElementElementwise/F_VN_MaxElementElementwise_ULINT

	{attribute 'TcIecLibraryType'}
	{attribute 'external_name' := 'F_VN_MaxElementElementwise_ULINT_GUID_09C9B808_951D_4EC2_FF90_CC002EBB19E0'}
	(* Gets the element wise maximum container element. *)
	FUNCTION F_VN_MaxElementElementwise_ULINT : HRESULT
	VAR_INPUT
		ipContainer	:	ITcVnContainer;	(* Source container *)
	END_VAR
	VAR_IN_OUT
		nMax	:	ULINT;	(* Returns the requested element *)
	END_VAR
	VAR_INPUT
		hrPrev	:	HRESULT;	(* HRESULT indicating the result of previous operations (If SUCCEEDED(hrPrev) equals false, no operation is executed.) *)
	END_VAR

END_FUNCTION

// Functions/Container Statistics/F_VN_MaxElementElementwise/F_VN_MaxElementElementwise_USINT

	{attribute 'TcIecLibraryType'}
	{attribute 'external_name' := 'F_VN_MaxElementElementwise_USINT_GUID_157B1579_B25E_4A20_EFC6_E977629AB2D4'}
	(* Gets the element wise maximum container element. *)
	FUNCTION F_VN_MaxElementElementwise_USINT : HRESULT
	VAR_INPUT
		ipContainer	:	ITcVnContainer;	(* Source container *)
	END_VAR
	VAR_IN_OUT
		nMax	:	USINT;	(* Returns the requested element *)
	END_VAR
	VAR_INPUT
		hrPrev	:	HRESULT;	(* HRESULT indicating the result of previous operations (If SUCCEEDED(hrPrev) equals false, no operation is executed.) *)
	END_VAR

END_FUNCTION

// Functions/Container Statistics/F_VN_MedianElementElementwise/F_VN_MedianElementElementwise_DINT

	{attribute 'TcIecLibraryType'}
	{attribute 'external_name' := 'F_VN_MedianElementElementwise_DINT_GUID_59346E04_1C02_48A3_E4F3_B292AF406D95'}
	(* Gets the element wise median container element. *)
	FUNCTION F_VN_MedianElementElementwise_DINT : HRESULT
	VAR_INPUT
		ipContainer	:	ITcVnContainer;	(* Source container *)
	END_VAR
	VAR_IN_OUT
		nMedian	:	DINT;	(* Returns the requested element *)
	END_VAR
	VAR_INPUT
		hrPrev	:	HRESULT;	(* HRESULT indicating the result of previous operations (If SUCCEEDED(hrPrev) equals false, no operation is executed.) *)
	END_VAR

END_FUNCTION

// Functions/Container Statistics/F_VN_MedianElementElementwise/F_VN_MedianElementElementwise_INT

	{attribute 'TcIecLibraryType'}
	{attribute 'external_name' := 'F_VN_MedianElementElementwise_INT_GUID_BB942F0C_1BA3_4DA8_E8D9_1E5175F12DE4'}
	(* Gets the element wise median container element. *)
	FUNCTION F_VN_MedianElementElementwise_INT : HRESULT
	VAR_INPUT
		ipContainer	:	ITcVnContainer;	(* Source container *)
	END_VAR
	VAR_IN_OUT
		nMedian	:	INT;	(* Returns the requested element *)
	END_VAR
	VAR_INPUT
		hrPrev	:	HRESULT;	(* HRESULT indicating the result of previous operations (If SUCCEEDED(hrPrev) equals false, no operation is executed.) *)
	END_VAR

END_FUNCTION

// Functions/Container Statistics/F_VN_MedianElementElementwise/F_VN_MedianElementElementwise_LREAL

	{attribute 'TcIecLibraryType'}
	{attribute 'external_name' := 'F_VN_MedianElementElementwise_LREAL_GUID_C5FFF627_63AA_4316_C79B_794D88DE6069'}
	(* Gets the element wise median container element. *)
	FUNCTION F_VN_MedianElementElementwise_LREAL : HRESULT
	VAR_INPUT
		ipContainer	:	ITcVnContainer;	(* Source container *)
	END_VAR
	VAR_IN_OUT
		fMedian	:	LREAL;	(* Returns the requested element *)
	END_VAR
	VAR_INPUT
		hrPrev	:	HRESULT;	(* HRESULT indicating the result of previous operations (If SUCCEEDED(hrPrev) equals false, no operation is executed.) *)
	END_VAR

END_FUNCTION

// Functions/Container Statistics/F_VN_MedianElementElementwise/F_VN_MedianElementElementwise_REAL

	{attribute 'TcIecLibraryType'}
	{attribute 'external_name' := 'F_VN_MedianElementElementwise_REAL_GUID_5140119F_67AB_4360_E0B7_EF95B24C8B21'}
	(* Gets the element wise median container element. *)
	FUNCTION F_VN_MedianElementElementwise_REAL : HRESULT
	VAR_INPUT
		ipContainer	:	ITcVnContainer;	(* Source container *)
	END_VAR
	VAR_IN_OUT
		fMedian	:	REAL;	(* Returns the requested element *)
	END_VAR
	VAR_INPUT
		hrPrev	:	HRESULT;	(* HRESULT indicating the result of previous operations (If SUCCEEDED(hrPrev) equals false, no operation is executed.) *)
	END_VAR

END_FUNCTION

// Functions/Container Statistics/F_VN_MedianElementElementwise/F_VN_MedianElementElementwise_SINT

	{attribute 'TcIecLibraryType'}
	{attribute 'external_name' := 'F_VN_MedianElementElementwise_SINT_GUID_D7F5B6FE_FDE8_47E2_CD7B_1BA54B747FCF'}
	(* Gets the element wise median container element. *)
	FUNCTION F_VN_MedianElementElementwise_SINT : HRESULT
	VAR_INPUT
		ipContainer	:	ITcVnContainer;	(* Source container *)
	END_VAR
	VAR_IN_OUT
		nMedian	:	SINT;	(* Returns the requested element *)
	END_VAR
	VAR_INPUT
		hrPrev	:	HRESULT;	(* HRESULT indicating the result of previous operations (If SUCCEEDED(hrPrev) equals false, no operation is executed.) *)
	END_VAR

END_FUNCTION

// Functions/Container Statistics/F_VN_MedianElementElementwise/F_VN_MedianElementElementwise_TcVnPoint2_DINT

	{attribute 'TcIecLibraryType'}
	{attribute 'external_name' := 'F_VN_MedianElementElementwise_TcVnPoint2_DINT_GUID_D3C7C4F5_BD25_4829_E89B_0BAD7D8EF0A2'}
	(* Gets the element wise median container element. *)
	FUNCTION F_VN_MedianElementElementwise_TcVnPoint2_DINT : HRESULT
	VAR_INPUT
		ipContainer	:	ITcVnContainer;	(* Source container *)
	END_VAR
	VAR_IN_OUT
		aMedian	:	TcVnPoint2_DINT;	(* Returns the requested element *)
	END_VAR
	VAR_INPUT
		hrPrev	:	HRESULT;	(* HRESULT indicating the result of previous operations (If SUCCEEDED(hrPrev) equals false, no operation is executed.) *)
	END_VAR

END_FUNCTION

// Functions/Container Statistics/F_VN_MedianElementElementwise/F_VN_MedianElementElementwise_TcVnPoint2_LREAL

	{attribute 'TcIecLibraryType'}
	{attribute 'external_name' := 'F_VN_MedianElementElementwise_TcVnPoint2_LREAL_GUID_28342F63_A38E_4FAC_F13F_8E42D8057A70'}
	(* Gets the element wise median container element. *)
	FUNCTION F_VN_MedianElementElementwise_TcVnPoint2_LREAL : HRESULT
	VAR_INPUT
		ipContainer	:	ITcVnContainer;	(* Source container *)
	END_VAR
	VAR_IN_OUT
		aMedian	:	TcVnPoint2_LREAL;	(* Returns the requested element *)
	END_VAR
	VAR_INPUT
		hrPrev	:	HRESULT;	(* HRESULT indicating the result of previous operations (If SUCCEEDED(hrPrev) equals false, no operation is executed.) *)
	END_VAR

END_FUNCTION

// Functions/Container Statistics/F_VN_MedianElementElementwise/F_VN_MedianElementElementwise_TcVnPoint2_REAL

	{attribute 'TcIecLibraryType'}
	{attribute 'external_name' := 'F_VN_MedianElementElementwise_TcVnPoint2_REAL_GUID_88CD9B3E_D013_4679_C20B_C7DC1CA7BB70'}
	(* Gets the element wise median container element. *)
	FUNCTION F_VN_MedianElementElementwise_TcVnPoint2_REAL : HRESULT
	VAR_INPUT
		ipContainer	:	ITcVnContainer;	(* Source container *)
	END_VAR
	VAR_IN_OUT
		aMedian	:	TcVnPoint2_REAL;	(* Returns the requested element *)
	END_VAR
	VAR_INPUT
		hrPrev	:	HRESULT;	(* HRESULT indicating the result of previous operations (If SUCCEEDED(hrPrev) equals false, no operation is executed.) *)
	END_VAR

END_FUNCTION

// Functions/Container Statistics/F_VN_MedianElementElementwise/F_VN_MedianElementElementwise_TcVnPoint3_LREAL

	{attribute 'TcIecLibraryType'}
	{attribute 'external_name' := 'F_VN_MedianElementElementwise_TcVnPoint3_LREAL_GUID_81D4DB37_DB25_48C2_F7DD_FBC8ACC6B9FB'}
	(* Gets the element wise median container element. *)
	FUNCTION F_VN_MedianElementElementwise_TcVnPoint3_LREAL : HRESULT
	VAR_INPUT
		ipContainer	:	ITcVnContainer;	(* Source container *)
	END_VAR
	VAR_IN_OUT
		aMedian	:	TcVnPoint3_LREAL;	(* Returns the requested element *)
	END_VAR
	VAR_INPUT
		hrPrev	:	HRESULT;	(* HRESULT indicating the result of previous operations (If SUCCEEDED(hrPrev) equals false, no operation is executed.) *)
	END_VAR

END_FUNCTION

// Functions/Container Statistics/F_VN_MedianElementElementwise/F_VN_MedianElementElementwise_TcVnPoint3_REAL

	{attribute 'TcIecLibraryType'}
	{attribute 'external_name' := 'F_VN_MedianElementElementwise_TcVnPoint3_REAL_GUID_05F1C071_8EAF_4B51_F843_6F556C41DB08'}
	(* Gets the element wise median container element. *)
	FUNCTION F_VN_MedianElementElementwise_TcVnPoint3_REAL : HRESULT
	VAR_INPUT
		ipContainer	:	ITcVnContainer;	(* Source container *)
	END_VAR
	VAR_IN_OUT
		aMedian	:	TcVnPoint3_REAL;	(* Returns the requested element *)
	END_VAR
	VAR_INPUT
		hrPrev	:	HRESULT;	(* HRESULT indicating the result of previous operations (If SUCCEEDED(hrPrev) equals false, no operation is executed.) *)
	END_VAR

END_FUNCTION

// Functions/Container Statistics/F_VN_MedianElementElementwise/F_VN_MedianElementElementwise_TcVnVector2_DINT

	{attribute 'TcIecLibraryType'}
	{attribute 'external_name' := 'F_VN_MedianElementElementwise_TcVnVector2_DINT_GUID_FED9DDAE_5E9C_4F0B_C5C7_8216CE609818'}
	(* Gets the element wise median container element. *)
	FUNCTION F_VN_MedianElementElementwise_TcVnVector2_DINT : HRESULT
	VAR_INPUT
		ipContainer	:	ITcVnContainer;	(* Source container *)
	END_VAR
	VAR_IN_OUT
		aMedian	:	TcVnVector2_DINT;	(* Returns the requested element *)
	END_VAR
	VAR_INPUT
		hrPrev	:	HRESULT;	(* HRESULT indicating the result of previous operations (If SUCCEEDED(hrPrev) equals false, no operation is executed.) *)
	END_VAR

END_FUNCTION

// Functions/Container Statistics/F_VN_MedianElementElementwise/F_VN_MedianElementElementwise_TcVnVector2_INT

	{attribute 'TcIecLibraryType'}
	{attribute 'external_name' := 'F_VN_MedianElementElementwise_TcVnVector2_INT_GUID_2B43DCE7_4BCE_4E23_FAEC_A94414AF5E35'}
	(* Gets the element wise median container element. *)
	FUNCTION F_VN_MedianElementElementwise_TcVnVector2_INT : HRESULT
	VAR_INPUT
		ipContainer	:	ITcVnContainer;	(* Source container *)
	END_VAR
	VAR_IN_OUT
		aMedian	:	TcVnVector2_INT;	(* Returns the requested element *)
	END_VAR
	VAR_INPUT
		hrPrev	:	HRESULT;	(* HRESULT indicating the result of previous operations (If SUCCEEDED(hrPrev) equals false, no operation is executed.) *)
	END_VAR

END_FUNCTION

// Functions/Container Statistics/F_VN_MedianElementElementwise/F_VN_MedianElementElementwise_TcVnVector2_REAL

	{attribute 'TcIecLibraryType'}
	{attribute 'external_name' := 'F_VN_MedianElementElementwise_TcVnVector2_REAL_GUID_F6775716_1AA9_4787_CD8F_41BDAB847EBA'}
	(* Gets the element wise median container element. *)
	FUNCTION F_VN_MedianElementElementwise_TcVnVector2_REAL : HRESULT
	VAR_INPUT
		ipContainer	:	ITcVnContainer;	(* Source container *)
	END_VAR
	VAR_IN_OUT
		aMedian	:	TcVnVector2_REAL;	(* Returns the requested element *)
	END_VAR
	VAR_INPUT
		hrPrev	:	HRESULT;	(* HRESULT indicating the result of previous operations (If SUCCEEDED(hrPrev) equals false, no operation is executed.) *)
	END_VAR

END_FUNCTION

// Functions/Container Statistics/F_VN_MedianElementElementwise/F_VN_MedianElementElementwise_TcVnVector2_SINT

	{attribute 'TcIecLibraryType'}
	{attribute 'external_name' := 'F_VN_MedianElementElementwise_TcVnVector2_SINT_GUID_8FB9F193_5BEB_4F5D_DED3_B5402A68C727'}
	(* Gets the element wise median container element. *)
	FUNCTION F_VN_MedianElementElementwise_TcVnVector2_SINT : HRESULT
	VAR_INPUT
		ipContainer	:	ITcVnContainer;	(* Source container *)
	END_VAR
	VAR_IN_OUT
		aMedian	:	TcVnVector2_SINT;	(* Returns the requested element *)
	END_VAR
	VAR_INPUT
		hrPrev	:	HRESULT;	(* HRESULT indicating the result of previous operations (If SUCCEEDED(hrPrev) equals false, no operation is executed.) *)
	END_VAR

END_FUNCTION

// Functions/Container Statistics/F_VN_MedianElementElementwise/F_VN_MedianElementElementwise_TcVnVector2_UINT

	{attribute 'TcIecLibraryType'}
	{attribute 'external_name' := 'F_VN_MedianElementElementwise_TcVnVector2_UINT_GUID_00C69F67_86DF_4C93_F206_4CFE453DB271'}
	(* Gets the element wise median container element. *)
	FUNCTION F_VN_MedianElementElementwise_TcVnVector2_UINT : HRESULT
	VAR_INPUT
		ipContainer	:	ITcVnContainer;	(* Source container *)
	END_VAR
	VAR_IN_OUT
		aMedian	:	TcVnVector2_UINT;	(* Returns the requested element *)
	END_VAR
	VAR_INPUT
		hrPrev	:	HRESULT;	(* HRESULT indicating the result of previous operations (If SUCCEEDED(hrPrev) equals false, no operation is executed.) *)
	END_VAR

END_FUNCTION

// Functions/Container Statistics/F_VN_MedianElementElementwise/F_VN_MedianElementElementwise_TcVnVector2_USINT

	{attribute 'TcIecLibraryType'}
	{attribute 'external_name' := 'F_VN_MedianElementElementwise_TcVnVector2_USINT_GUID_55EEF251_DC7E_4CE5_C2BE_4BECB336F045'}
	(* Gets the element wise median container element. *)
	FUNCTION F_VN_MedianElementElementwise_TcVnVector2_USINT : HRESULT
	VAR_INPUT
		ipContainer	:	ITcVnContainer;	(* Source container *)
	END_VAR
	VAR_IN_OUT
		aMedian	:	TcVnVector2_USINT;	(* Returns the requested element *)
	END_VAR
	VAR_INPUT
		hrPrev	:	HRESULT;	(* HRESULT indicating the result of previous operations (If SUCCEEDED(hrPrev) equals false, no operation is executed.) *)
	END_VAR

END_FUNCTION

// Functions/Container Statistics/F_VN_MedianElementElementwise/F_VN_MedianElementElementwise_TcVnVector3_INT

	{attribute 'TcIecLibraryType'}
	{attribute 'external_name' := 'F_VN_MedianElementElementwise_TcVnVector3_INT_GUID_3C483EB7_00C7_423B_F0A3_E0A24D16B7DD'}
	(* Gets the element wise median container element. *)
	FUNCTION F_VN_MedianElementElementwise_TcVnVector3_INT : HRESULT
	VAR_INPUT
		ipContainer	:	ITcVnContainer;	(* Source container *)
	END_VAR
	VAR_IN_OUT
		aMedian	:	TcVnVector3_INT;	(* Returns the requested element *)
	END_VAR
	VAR_INPUT
		hrPrev	:	HRESULT;	(* HRESULT indicating the result of previous operations (If SUCCEEDED(hrPrev) equals false, no operation is executed.) *)
	END_VAR

END_FUNCTION

// Functions/Container Statistics/F_VN_MedianElementElementwise/F_VN_MedianElementElementwise_TcVnVector3_REAL

	{attribute 'TcIecLibraryType'}
	{attribute 'external_name' := 'F_VN_MedianElementElementwise_TcVnVector3_REAL_GUID_3E07A55F_20E7_4EF6_C8B3_061AE81D4F55'}
	(* Gets the element wise median container element. *)
	FUNCTION F_VN_MedianElementElementwise_TcVnVector3_REAL : HRESULT
	VAR_INPUT
		ipContainer	:	ITcVnContainer;	(* Source container *)
	END_VAR
	VAR_IN_OUT
		aMedian	:	TcVnVector3_REAL;	(* Returns the requested element *)
	END_VAR
	VAR_INPUT
		hrPrev	:	HRESULT;	(* HRESULT indicating the result of previous operations (If SUCCEEDED(hrPrev) equals false, no operation is executed.) *)
	END_VAR

END_FUNCTION

// Functions/Container Statistics/F_VN_MedianElementElementwise/F_VN_MedianElementElementwise_TcVnVector3_SINT

	{attribute 'TcIecLibraryType'}
	{attribute 'external_name' := 'F_VN_MedianElementElementwise_TcVnVector3_SINT_GUID_E1A93D89_F678_42E3_DEA5_48C534D9F1A9'}
	(* Gets the element wise median container element. *)
	FUNCTION F_VN_MedianElementElementwise_TcVnVector3_SINT : HRESULT
	VAR_INPUT
		ipContainer	:	ITcVnContainer;	(* Source container *)
	END_VAR
	VAR_IN_OUT
		aMedian	:	TcVnVector3_SINT;	(* Returns the requested element *)
	END_VAR
	VAR_INPUT
		hrPrev	:	HRESULT;	(* HRESULT indicating the result of previous operations (If SUCCEEDED(hrPrev) equals false, no operation is executed.) *)
	END_VAR

END_FUNCTION

// Functions/Container Statistics/F_VN_MedianElementElementwise/F_VN_MedianElementElementwise_TcVnVector3_UINT

	{attribute 'TcIecLibraryType'}
	{attribute 'external_name' := 'F_VN_MedianElementElementwise_TcVnVector3_UINT_GUID_D84167C4_BF7A_4850_CE92_FF22134CE87D'}
	(* Gets the element wise median container element. *)
	FUNCTION F_VN_MedianElementElementwise_TcVnVector3_UINT : HRESULT
	VAR_INPUT
		ipContainer	:	ITcVnContainer;	(* Source container *)
	END_VAR
	VAR_IN_OUT
		aMedian	:	TcVnVector3_UINT;	(* Returns the requested element *)
	END_VAR
	VAR_INPUT
		hrPrev	:	HRESULT;	(* HRESULT indicating the result of previous operations (If SUCCEEDED(hrPrev) equals false, no operation is executed.) *)
	END_VAR

END_FUNCTION

// Functions/Container Statistics/F_VN_MedianElementElementwise/F_VN_MedianElementElementwise_TcVnVector3_USINT

	{attribute 'TcIecLibraryType'}
	{attribute 'external_name' := 'F_VN_MedianElementElementwise_TcVnVector3_USINT_GUID_7C117060_F216_40BE_C1D4_042D9C61F407'}
	(* Gets the element wise median container element. *)
	FUNCTION F_VN_MedianElementElementwise_TcVnVector3_USINT : HRESULT
	VAR_INPUT
		ipContainer	:	ITcVnContainer;	(* Source container *)
	END_VAR
	VAR_IN_OUT
		aMedian	:	TcVnVector3_USINT;	(* Returns the requested element *)
	END_VAR
	VAR_INPUT
		hrPrev	:	HRESULT;	(* HRESULT indicating the result of previous operations (If SUCCEEDED(hrPrev) equals false, no operation is executed.) *)
	END_VAR

END_FUNCTION

// Functions/Container Statistics/F_VN_MedianElementElementwise/F_VN_MedianElementElementwise_TcVnVector4_DINT

	{attribute 'TcIecLibraryType'}
	{attribute 'external_name' := 'F_VN_MedianElementElementwise_TcVnVector4_DINT_GUID_1F334392_F839_45F8_CB91_66F65DF87769'}
	(* Gets the element wise median container element. *)
	FUNCTION F_VN_MedianElementElementwise_TcVnVector4_DINT : HRESULT
	VAR_INPUT
		ipContainer	:	ITcVnContainer;	(* Source container *)
	END_VAR
	VAR_IN_OUT
		aMedian	:	TcVnVector4_DINT;	(* Returns the requested element *)
	END_VAR
	VAR_INPUT
		hrPrev	:	HRESULT;	(* HRESULT indicating the result of previous operations (If SUCCEEDED(hrPrev) equals false, no operation is executed.) *)
	END_VAR

END_FUNCTION

